LIN {X 0,Y 253.116,Z 526.81,A -85,B 0,C 180,E1 17086.147,E2 17086.147} C_VEL
LIN {X 0,Y 253.751,Z 526.81,A -85,B 0,C 180,E1 17093.136,E2 17093.136} C_VEL
LIN {X 0,Y 254.471,Z 526.81,A -85,B 0,C 180,E1 17099.989,E2 17099.989} C_VEL
LIN {X 0,Y 253.748,Z 526.81,A -85,B 0,C 180,E1 17106.843,E2 17106.843} C_VEL
LIN {X 0,Y 253.12,Z 526.81,A -85,B 0,C 180,E1 17113.832,E2 17113.832} C_VEL
LIN {X 0,Y 252.62,Z 526.81,A -85,B 0,C 180,E1 17121.064,E2 17121.064} C_VEL
LIN {X 0,Y 252.194,Z 526.81,A -85,B 0,C 180,E1 17128.69,E2 17128.69} C_VEL
LIN {X 0,Y 251.705,Z 526.81,A -85,B 0,C 180,E1 17136.964,E2 17136.964} C_VEL
LIN {X 0,Y 251.565,Z 526.81,A -85,B 0,C 180,E1 17146.221,E2 17146.221} C_VEL
LIN {X 0,Y 251.958,Z 526.81,A -85,B 0,C 180,E1 17150.844,E2 17150.844} C_VEL
LIN {X 0,Y 270.86,Z 591.901,A -85,B 0,C 180,E1 17154.954,E2 17154.954} C_VEL
LIN {X 0,Y 272.504,Z 601.249,A -85,B 0,C 180,E1 17155.665,E2 17155.665} C_VEL
LIN {X 0,Y 268.172,Z 634.394,A -85,B 0,C 180,E1 17158.572,E2 17158.572} C_VEL
LIN {X 0,Y 263.468,Z 664.052,A -85,B 0,C 180,E1 17162.639,E2 17162.639} C_VEL
LIN {X 0,Y 259.639,Z 689.343,A -85,B 0,C 180,E1 17167.736,E2 17167.736} C_VEL
LIN {X 0,Y 257.402,Z 710.001,A -85,B 0,C 180,E1 17173.784,E2 17173.784} C_VEL
LIN {X 0,Y 257.027,Z 723.846,A -85,B 0,C 180,E1 17179.829,E2 17179.829} C_VEL
LIN {X 0,Y 257.514,Z 731.331,A -85,B 0,C 180,E1 17184.948,E2 17184.948} C_VEL
LIN {X 0,Y 257.788,Z 735.161,A -85,B 0,C 180,E1 17190.008,E2 17190.008} C_VEL
LIN {X 0,Y 256.526,Z 734.875,A -85,B 0,C 180,E1 17196.787,E2 17196.787} C_VEL
LIN {X 0,Y 256.215,Z 728.457,A -85,B 0,C 180,E1 17204.554,E2 17204.554} C_VEL
LIN {X 0,Y 259.476,Z 716.032,A -85,B 0,C 180,E1 17212.298,E2 17212.298} C_VEL
LIN {X 0,Y 267.703,Z 697.17,A -85,B 0,C 180,E1 17219.671,E2 17219.671} C_VEL
LIN {X 0,Y 278.883,Z 674.315,A -85,B 0,C 180,E1 17225.604,E2 17225.604} C_VEL
LIN {X 0,Y 292.583,Z 646.621,A -85,B 0,C 180,E1 17230.314,E2 17230.314} C_VEL
LIN {X 0,Y 306.811,Z 613.528,A -85,B 0,C 180,E1 17234.03,E2 17234.03} C_VEL
LIN {X 0,Y 305.668,Z 605.43,A -85,B 0,C 180,E1 17237.281,E2 17237.281} C_VEL
LIN {X 0,Y 304.554,Z 603.17,A -85,B 0,C 180,E1 17239.752,E2 17239.752} C_VEL
LIN {X 0,Y 303.432,Z 604.168,A -85,B 0,C 180,E1 17243.231,E2 17243.231} C_VEL
LIN {X 0,Y 301.963,Z 610.894,A -85,B 0,C 180,E1 17246.944,E2 17246.944} C_VEL
LIN {X 0,Y 299.587,Z 618.107,A -85,B 0,C 180,E1 17248.987,E2 17248.987} C_VEL
LIN {X 0,Y 287.255,Z 640.013,A -85,B 0,C 180,E1 17253.395,E2 17253.395} C_VEL
LIN {X 0,Y 276.783,Z 655.626,A -85,B 0,C 180,E1 17258.428,E2 17258.428} C_VEL
LIN {X 0,Y 273.369,Z 659.975,A -85,B 0,C 180,E1 17260.458,E2 17260.458} C_VEL
LIN {X 0,Y 265.293,Z 666.359,A -85,B 0,C 180,E1 17263.486,E2 17263.486} C_VEL
LIN {X 0,Y 258.207,Z 669.931,A -85,B 0,C 180,E1 17266.346,E2 17266.346} C_VEL
LIN {X 0,Y 257.614,Z 670.127,A -85,B 0,C 180,E1 17266.81,E2 17266.81} C_VEL
LIN {X 0,Y 254.828,Z 671.039,A -85,B 0,C 180,E1 17269.744,E2 17269.744} C_VEL
LIN {X 0,Y 251.775,Z 669.41,A -85,B 0,C 180,E1 17274.836,E2 17274.836} C_VEL
LIN {X 0,Y 249.796,Z 662.54,A -85,B 0,C 180,E1 17280.912,E2 17280.912} C_VEL
LIN {X 0,Y 249.682,Z 649.701,A -85,B 0,C 180,E1 17286.976,E2 17286.976} C_VEL
LIN {X 0,Y 250.995,Z 630.908,A -85,B 0,C 180,E1 17292.641,E2 17292.641} C_VEL
LIN {X 0,Y 253.302,Z 607.549,A -85,B 0,C 180,E1 17297.4,E2 17297.4} C_VEL
LIN {X 0,Y 255.637,Z 580.367,A -85,B 0,C 180,E1 17301.17,E2 17301.17} C_VEL
LIN {X 0,Y 249.736,Z 549.406,A -85,B 0,C 180,E1 17304.37,E2 17304.37} C_VEL
LIN {X 0,Y 244.584,Z 526.81,A -85,B 0,C 180,E1 17306.183,E2 17306.183} C_VEL
LIN {X 0,Y 243.774,Z 526.81,A -85,B 0,C 180,E1 17316.141,E2 17316.141} C_VEL
LIN {X 0,Y 243.692,Z 526.81,A -85,B 0,C 180,E1 17323.125,E2 17323.125} C_VEL
LIN {X 0,Y 243.814,Z 526.81,A -85,B 0,C 180,E1 17331.601,E2 17331.601} C_VEL
LIN {X 0,Y 244.154,Z 526.81,A -85,B 0,C 180,E1 17340.265,E2 17340.265} C_VEL
LIN {X 0,Y 244.619,Z 526.81,A -85,B 0,C 180,E1 17348.212,E2 17348.212} C_VEL
LIN {X 0,Y 245.142,Z 526.81,A -85,B 0,C 180,E1 17355.688,E2 17355.688} C_VEL
LIN {X 0,Y 245.771,Z 526.81,A -85,B 0,C 180,E1 17362.914,E2 17362.914} C_VEL
LIN {X 0,Y 246.595,Z 526.81,A -85,B 0,C 180,E1 17369.992,E2 17369.992} C_VEL
LIN {X 0,Y 245.582,Z 526.81,A -85,B 0,C 180,E1 17379.399,E2 17379.399} C_VEL
LIN {X 0,Y 244.892,Z 526.81,A -85,B 0,C 180,E1 17387.998,E2 17387.998} C_VEL
LIN {X 0,Y 244.381,Z 526.81,A -85,B 0,C 180,E1 17395.692,E2 17395.692} C_VEL
LIN {X 0,Y 243.826,Z 526.81,A -85,B 0,C 180,E1 17403.967,E2 17403.967} C_VEL
LIN {X 0,Y 243.67,Z 526.81,A -85,B 0,C 180,E1 17413.106,E2 17413.106} C_VEL
LIN {X 0,Y 243.782,Z 526.81,A -85,B 0,C 180,E1 17421.594,E2 17421.594} C_VEL
LIN {X 0,Y 244.125,Z 526.81,A -85,B 0,C 180,E1 17430.243,E2 17430.243} C_VEL
LIN {X 0,Y 244.587,Z 526.81,A -85,B 0,C 180,E1 17438.186,E2 17438.186} C_VEL
LIN {X 0,Y 245.163,Z 526.81,A -85,B 0,C 180,E1 17445.688,E2 17445.688} C_VEL
LIN {X 0,Y 245.795,Z 526.81,A -85,B 0,C 180,E1 17452.913,E2 17452.913} C_VEL
LIN {X 0,Y 246.561,Z 526.81,A -85,B 0,C 180,E1 17459.989,E2 17459.989} C_VEL
LIN {X 0,Y 245.521,Z 526.81,A -85,B 0,C 180,E1 17469.413,E2 17469.413} C_VEL
LIN {X 0,Y 244.876,Z 526.81,A -85,B 0,C 180,E1 17477.996,E2 17477.996} C_VEL
LIN {X 0,Y 244.366,Z 526.81,A -85,B 0,C 180,E1 17485.69,E2 17485.69} C_VEL
LIN {X 0,Y 243.887,Z 526.81,A -85,B 0,C 180,E1 17493.953,E2 17493.953} C_VEL
LIN {X 0,Y 243.613,Z 526.81,A -85,B 0,C 180,E1 17503.112,E2 17503.112} C_VEL
LIN {X 0,Y 243.978,Z 526.81,A -85,B 0,C 180,E1 17510.328,E2 17510.328} C_VEL
LIN {X 0,Y 262.39,Z 590.644,A -85,B 0,C 180,E1 17514.439,E2 17514.439} C_VEL
LIN {X 0,Y 264.827,Z 601.026,A -85,B 0,C 180,E1 17515.279,E2 17515.279} C_VEL
LIN {X 0,Y 260.497,Z 633.255,A -85,B 0,C 180,E1 17518.198,E2 17518.198} C_VEL
LIN {X 0,Y 255.668,Z 663.218,A -85,B 0,C 180,E1 17522.425,E2 17522.425} C_VEL
LIN {X 0,Y 251.929,Z 687.654,A -85,B 0,C 180,E1 17527.481,E2 17527.481} C_VEL
LIN {X 0,Y 249.615,Z 708.493,A -85,B 0,C 180,E1 17533.716,E2 17533.716} C_VEL
LIN {X 0,Y 249.295,Z 723.223,A -85,B 0,C 180,E1 17540.394,E2 17540.394} C_VEL
LIN {X 0,Y 249.892,Z 731.257,A -85,B 0,C 180,E1 17546.535,E2 17546.535} C_VEL
LIN {X 0,Y 250.046,Z 733.566,A -85,B 0,C 180,E1 17550.008,E2 17550.008} C_VEL
LIN {X 0,Y 248.649,Z 733.566,A -85,B 0,C 180,E1 17557.003,E2 17557.003} C_VEL
LIN {X 0,Y 248.426,Z 727.533,A -85,B 0,C 180,E1 17565.021,E2 17565.021} C_VEL
LIN {X 0,Y 252.03,Z 715.545,A -85,B 0,C 180,E1 17572.994,E2 17572.994} C_VEL
LIN {X 0,Y 260.787,Z 697.428,A -85,B 0,C 180,E1 17580.54,E2 17580.54} C_VEL
LIN {X 0,Y 273.2,Z 674.491,A -85,B 0,C 180,E1 17586.794,E2 17586.794} C_VEL
LIN {X 0,Y 288.54,Z 646.199,A -85,B 0,C 180,E1 17591.75,E2 17591.75} C_VEL
LIN {X 0,Y 302.164,Z 617.648,A -85,B 0,C 180,E1 17595.064,E2 17595.064} C_VEL
LIN {X 0,Y 301.617,Z 612.201,A -85,B 0,C 180,E1 17597.46,E2 17597.46} C_VEL
LIN {X 0,Y 300.866,Z 610.491,A -85,B 0,C 180,E1 17599.155,E2 17599.155} C_VEL
LIN {X 0,Y 299.468,Z 610.666,A -85,B 0,C 180,E1 17602.662,E2 17602.662} C_VEL
LIN {X 0,Y 297.762,Z 615.675,A -85,B 0,C 180,E1 17606.003,E2 17606.003} C_VEL
LIN {X 0,Y 295.36,Z 621.611,A -85,B 0,C 180,E1 17607.883,E2 17607.883} C_VEL
LIN {X 0,Y 281.88,Z 643.133,A -85,B 0,C 180,E1 17612.414,E2 17612.414} C_VEL
LIN {X 0,Y 270.332,Z 658.41,A -85,B 0,C 180,E1 17617.671,E2 17617.671} C_VEL
LIN {X 0,Y 261.607,Z 667.374,A -85,B 0,C 180,E1 17623.191,E2 17623.191} C_VEL
LIN {X 0,Y 257.614,Z 670.127,A -85,B 0,C 180,E1 17626.81,E2 17626.81} C_VEL
LIN {X 0,Y 250.472,Z 671.806,A -85,B 0,C 180,E1 17630.393,E2 17630.393} C_VEL
LIN {X 0,Y 244.609,Z 671.157,A -85,B 0,C 180,E1 17633.65,E2 17633.65} C_VEL
LIN {X 0,Y 244.257,Z 670.821,A -85,B 0,C 180,E1 17634.149,E2 17634.149} C_VEL
LIN {X 0,Y 242.145,Z 664.48,A -85,B 0,C 180,E1 17640.011,E2 17640.011} C_VEL
LIN {X 0,Y 241.743,Z 651.942,A -85,B 0,C 180,E1 17646.303,E2 17646.303} C_VEL
LIN {X 0,Y 242.942,Z 633.679,A -85,B 0,C 180,E1 17652.153,E2 17652.153} C_VEL
LIN {X 0,Y 245.326,Z 609.376,A -85,B 0,C 180,E1 17657.362,E2 17657.362} C_VEL
LIN {X 0,Y 247.856,Z 581.525,A -85,B 0,C 180,E1 17661.394,E2 17661.394} C_VEL
LIN {X 0,Y 242.234,Z 551.6,A -85,B 0,C 180,E1 17664.615,E2 17664.615} C_VEL
LIN {X 0,Y 236.604,Z 526.81,A -85,B 0,C 180,E1 17666.623,E2 17666.623} C_VEL
LIN {X 0,Y 235.859,Z 526.81,A -85,B 0,C 180,E1 17675.304,E2 17675.304} C_VEL
LIN {X 0,Y 235.758,Z 526.81,A -85,B 0,C 180,E1 17679.969,E2 17679.969} C_VEL
LIN {X 0,Y 235.687,Z 526.81,A -85,B 0,C 180,E1 17685.025,E2 17685.025} C_VEL
LIN {X 0,Y 235.788,Z 526.81,A -85,B 0,C 180,E1 17690.418,E2 17690.418} C_VEL
LIN {X 0,Y 236.039,Z 526.81,A -85,B 0,C 180,E1 17699.115,E2 17699.115} C_VEL
LIN {X 0,Y 236.578,Z 526.81,A -85,B 0,C 180,E1 17707.409,E2 17707.409} C_VEL
LIN {X 0,Y 237.14,Z 526.81,A -85,B 0,C 180,E1 17715.194,E2 17715.194} C_VEL
LIN {X 0,Y 237.838,Z 526.81,A -85,B 0,C 180,E1 17722.677,E2 17722.677} C_VEL
LIN {X 0,Y 238.683,Z 526.81,A -85,B 0,C 180,E1 17729.991,E2 17729.991} C_VEL
LIN {X 0,Y 237.903,Z 526.81,A -85,B 0,C 180,E1 17737.304,E2 17737.304} C_VEL
LIN {X 0,Y 237,Z 526.81,A -85,B 0,C 180,E1 17746.581,E2 17746.581} C_VEL
LIN {X 0,Y 236.376,Z 526.81,A -85,B 0,C 180,E1 17756.247,E2 17756.247} C_VEL
LIN {X 0,Y 235.843,Z 526.81,A -85,B 0,C 180,E1 17765.284,E2 17765.284} C_VEL
LIN {X 0,Y 235.732,Z 526.81,A -85,B 0,C 180,E1 17769.951,E2 17769.951} C_VEL
LIN {X 0,Y 235.641,Z 526.81,A -85,B 0,C 180,E1 17775.013,E2 17775.013} C_VEL
LIN {X 0,Y 235.753,Z 526.81,A -85,B 0,C 180,E1 17780.4,E2 17780.4} C_VEL
LIN {X 0,Y 236.014,Z 526.81,A -85,B 0,C 180,E1 17789.111,E2 17789.111} C_VEL
LIN {X 0,Y 236.549,Z 526.81,A -85,B 0,C 180,E1 17797.405,E2 17797.405} C_VEL
LIN {X 0,Y 237.156,Z 526.81,A -85,B 0,C 180,E1 17805.194,E2 17805.194} C_VEL
LIN {X 0,Y 237.856,Z 526.81,A -85,B 0,C 180,E1 17812.675,E2 17812.675} C_VEL
LIN {X 0,Y 238.65,Z 526.81,A -85,B 0,C 180,E1 17819.989,E2 17819.989} C_VEL
LIN {X 0,Y 237.851,Z 526.81,A -85,B 0,C 180,E1 17827.303,E2 17827.303} C_VEL
LIN {X 0,Y 236.972,Z 526.81,A -85,B 0,C 180,E1 17836.619,E2 17836.619} C_VEL
LIN {X 0,Y 236.367,Z 526.81,A -85,B 0,C 180,E1 17846.282,E2 17846.282} C_VEL
LIN {X 0,Y 235.869,Z 526.81,A -85,B 0,C 180,E1 17855.274,E2 17855.274} C_VEL
LIN {X 0,Y 235.717,Z 526.81,A -85,B 0,C 180,E1 17859.948,E2 17859.948} C_VEL
LIN {X 0,Y 236.054,Z 527.414,A -85,B 0,C 180,E1 17869.796,E2 17869.796} C_VEL
LIN {X 0,Y 254.001,Z 589.667,A -85,B 0,C 180,E1 17873.938,E2 17873.938} C_VEL
LIN {X 0,Y 256.935,Z 602.437,A -85,B 0,C 180,E1 17875.009,E2 17875.009} C_VEL
LIN {X 0,Y 252.462,Z 634.482,A -85,B 0,C 180,E1 17878.105,E2 17878.105} C_VEL
LIN {X 0,Y 247.649,Z 663.805,A -85,B 0,C 180,E1 17882.485,E2 17882.485} C_VEL
LIN {X 0,Y 243.964,Z 687.652,A -85,B 0,C 180,E1 17887.668,E2 17887.668} C_VEL
LIN {X 0,Y 241.779,Z 708.126,A -85,B 0,C 180,E1 17894.108,E2 17894.108} C_VEL
LIN {X 0,Y 241.612,Z 722.544,A -85,B 0,C 180,E1 17900.995,E2 17900.995} C_VEL
LIN {X 0,Y 242.166,Z 729.412,A -85,B 0,C 180,E1 17906.424,E2 17906.424} C_VEL
LIN {X 0,Y 242.195,Z 732.019,A -85,B 0,C 180,E1 17910.32,E2 17910.32} C_VEL
LIN {X 0,Y 240.779,Z 732.236,A -85,B 0,C 180,E1 17917.233,E2 17917.233} C_VEL
LIN {X 0,Y 240.481,Z 727.454,A -85,B 0,C 180,E1 17924.595,E2 17924.595} C_VEL
LIN {X 0,Y 243.909,Z 716.681,A -85,B 0,C 180,E1 17932.837,E2 17932.837} C_VEL
LIN {X 0,Y 252.66,Z 700.014,A -85,B 0,C 180,E1 17940.631,E2 17940.631} C_VEL
LIN {X 0,Y 265.669,Z 678.147,A -85,B 0,C 180,E1 17947.257,E2 17947.257} C_VEL
LIN {X 0,Y 281.256,Z 652.198,A -85,B 0,C 180,E1 17952.301,E2 17952.301} C_VEL
LIN {X 0,Y 297.525,Z 622.132,A -85,B 0,C 180,E1 17956.037,E2 17956.037} C_VEL
LIN {X 0,Y 296.944,Z 617.891,A -85,B 0,C 180,E1 17958.497,E2 17958.497} C_VEL
LIN {X 0,Y 295.31,Z 617.241,A -85,B 0,C 180,E1 17962.044,E2 17962.044} C_VEL
LIN {X 0,Y 294.076,Z 619.565,A -85,B 0,C 180,E1 17964.432,E2 17964.432} C_VEL
LIN {X 0,Y 291.828,Z 624.383,A -85,B 0,C 180,E1 17966.558,E2 17966.558} C_VEL
LIN {X 0,Y 276.637,Z 646.313,A -85,B 0,C 180,E1 17971.399,E2 17971.399} C_VEL
LIN {X 0,Y 263.377,Z 661.863,A -85,B 0,C 180,E1 17977.18,E2 17977.18} C_VEL
LIN {X 0,Y 254.405,Z 669.729,A -85,B 0,C 180,E1 17982.7,E2 17982.7} C_VEL
LIN {X 0,Y 247.225,Z 672.621,A -85,B 0,C 180,E1 17989.425,E2 17989.425} C_VEL
LIN {X 0,Y 244.257,Z 670.821,A -85,B 0,C 180,E1 17994.149,E2 17994.149} C_VEL
LIN {X 0,Y 240.44,Z 668.494,A -85,B 0,C 180,E1 17997.074,E2 17997.074} C_VEL
LIN {X 0,Y 234.043,Z 662.72,A -85,B 0,C 180,E1 18001.393,E2 18001.393} C_VEL
LIN {X 0,Y 233.892,Z 661.818,A -85,B 0,C 180,E1 18001.886,E2 18001.886} C_VEL
LIN {X 0,Y 234.108,Z 646.79,A -85,B 0,C 180,E1 18008.378,E2 18008.378} C_VEL
LIN {X 0,Y 235.885,Z 625.302,A -85,B 0,C 180,E1 18014.413,E2 18014.413} C_VEL
LIN {X 0,Y 238.682,Z 598.201,A -85,B 0,C 180,E1 18019.464,E2 18019.464} C_VEL
LIN {X 0,Y 239.663,Z 580.078,A -85,B 0,C 180,E1 18021.919,E2 18021.919} C_VEL
LIN {X 0,Y 233.767,Z 549.81,A -85,B 0,C 180,E1 18025.2,E2 18025.2} C_VEL
LIN {X 0,Y 228.564,Z 526.81,A -85,B 0,C 180,E1 18027.075,E2 18027.075} C_VEL
LIN {X 0,Y 227.761,Z 526.81,A -85,B 0,C 180,E1 18037.073,E2 18037.073} C_VEL
LIN {X 0,Y 227.633,Z 526.81,A -85,B 0,C 180,E1 18047.039,E2 18047.039} C_VEL
LIN {X 0,Y 227.805,Z 526.81,A -85,B 0,C 180,E1 18053.25,E2 18053.25} C_VEL
LIN {X 0,Y 228.25,Z 526.81,A -85,B 0,C 180,E1 18062.323,E2 18062.323} C_VEL
LIN {X 0,Y 228.83,Z 526.81,A -85,B 0,C 180,E1 18070.671,E2 18070.671} C_VEL
LIN {X 0,Y 229.467,Z 526.81,A -85,B 0,C 180,E1 18078.574,E2 18078.574} C_VEL
LIN {X 0,Y 230.339,Z 526.81,A -85,B 0,C 180,E1 18086.222,E2 18086.222} C_VEL
LIN {X 0,Y 230.771,Z 526.81,A -85,B 0,C 180,E1 18089.991,E2 18089.991} C_VEL
LIN {X 0,Y 229.757,Z 526.81,A -85,B 0,C 180,E1 18098.647,E2 18098.647} C_VEL
LIN {X 0,Y 229.219,Z 526.81,A -85,B 0,C 180,E1 18105.311,E2 18105.311} C_VEL
LIN {X 0,Y 228.547,Z 526.81,A -85,B 0,C 180,E1 18113.411,E2 18113.411} C_VEL
LIN {X 0,Y 228.011,Z 526.81,A -85,B 0,C 180,E1 18122.078,E2 18122.078} C_VEL
LIN {X 0,Y 227.596,Z 526.81,A -85,B 0,C 180,E1 18131.689,E2 18131.689} C_VEL
LIN {X 0,Y 227.599,Z 526.81,A -85,B 0,C 180,E1 18138.287,E2 18138.287} C_VEL
LIN {X 0,Y 228.03,Z 526.81,A -85,B 0,C 180,E1 18147.903,E2 18147.903} C_VEL
LIN {X 0,Y 228.639,Z 526.81,A -85,B 0,C 180,E1 18157.962,E2 18157.962} C_VEL
LIN {X 0,Y 229.171,Z 526.81,A -85,B 0,C 180,E1 18164.665,E2 18164.665} C_VEL
LIN {X 0,Y 229.89,Z 526.81,A -85,B 0,C 180,E1 18172.42,E2 18172.42} C_VEL
LIN {X 0,Y 230.737,Z 526.81,A -85,B 0,C 180,E1 18179.988,E2 18179.988} C_VEL
LIN {X 0,Y 229.698,Z 526.81,A -85,B 0,C 180,E1 18188.668,E2 18188.668} C_VEL
LIN {X 0,Y 229.181,Z 526.81,A -85,B 0,C 180,E1 18195.31,E2 18195.31} C_VEL
LIN {X 0,Y 228.57,Z 526.81,A -85,B 0,C 180,E1 18203.405,E2 18203.405} C_VEL
LIN {X 0,Y 228.062,Z 526.81,A -85,B 0,C 180,E1 18212.065,E2 18212.065} C_VEL
LIN {X 0,Y 227.577,Z 526.81,A -85,B 0,C 180,E1 18221.687,E2 18221.687} C_VEL
LIN {X 0,Y 228.027,Z 527.128,A -85,B 0,C 180,E1 18229.188,E2 18229.188} C_VEL
LIN {X 0,Y 245.878,Z 589.566,A -85,B 0,C 180,E1 18233.502,E2 18233.502} C_VEL
LIN {X 0,Y 248.948,Z 604.366,A -85,B 0,C 180,E1 18234.8,E2 18234.8} C_VEL
LIN {X 0,Y 244.204,Z 637.001,A -85,B 0,C 180,E1 18238.207,E2 18238.207} C_VEL
LIN {X 0,Y 239.241,Z 666.623,A -85,B 0,C 180,E1 18243.004,E2 18243.004} C_VEL
LIN {X 0,Y 235.498,Z 691.165,A -85,B 0,C 180,E1 18248.889,E2 18248.889} C_VEL
LIN {X 0,Y 233.835,Z 709.815,A -85,B 0,C 180,E1 18255.424,E2 18255.424} C_VEL
LIN {X 0,Y 234.122,Z 723.122,A -85,B 0,C 180,E1 18262.577,E2 18262.577} C_VEL
LIN {X 0,Y 234.468,Z 729.027,A -85,B 0,C 180,E1 18268.159,E2 18268.159} C_VEL
LIN {X 0,Y 233.648,Z 731.198,A -85,B 0,C 180,E1 18273.724,E2 18273.724} C_VEL
LIN {X 0,Y 232.518,Z 729.191,A -85,B 0,C 180,E1 18281.274,E2 18281.274} C_VEL
LIN {X 0,Y 234.315,Z 721.136,A -85,B 0,C 180,E1 18290.077,E2 18290.077} C_VEL
LIN {X 0,Y 241.774,Z 706.72,A -85,B 0,C 180,E1 18298.779,E2 18298.779} C_VEL
LIN {X 0,Y 254.953,Z 686.263,A -85,B 0,C 180,E1 18306.442,E2 18306.442} C_VEL
LIN {X 0,Y 271.119,Z 662.206,A -85,B 0,C 180,E1 18312.088,E2 18312.088} C_VEL
LIN {X 0,Y 288.988,Z 633.302,A -85,B 0,C 180,E1 18316.368,E2 18316.368} C_VEL
LIN {X 0,Y 292.782,Z 626.559,A -85,B 0,C 180,E1 18317.136,E2 18317.136} C_VEL
LIN {X 0,Y 292.781,Z 625.361,A -85,B 0,C 180,E1 18317.772,E2 18317.772} C_VEL
LIN {X 0,Y 291.058,Z 623.729,A -85,B 0,C 180,E1 18321.388,E2 18321.388} C_VEL
LIN {X 0,Y 289.673,Z 625.406,A -85,B 0,C 180,E1 18323.833,E2 18323.833} C_VEL
LIN {X 0,Y 287.636,Z 628.846,A -85,B 0,C 180,E1 18325.549,E2 18325.549} C_VEL
LIN {X 0,Y 271.51,Z 649.614,A -85,B 0,C 180,E1 18330.349,E2 18330.349} C_VEL
LIN {X 0,Y 258.222,Z 663.596,A -85,B 0,C 180,E1 18335.78,E2 18335.78} C_VEL
LIN {X 0,Y 247.218,Z 672.025,A -85,B 0,C 180,E1 18342.181,E2 18342.181} C_VEL
LIN {X 0,Y 239.626,Z 674.161,A -85,B 0,C 180,E1 18349.085,E2 18349.085} C_VEL
LIN {X 0,Y 236.195,Z 671.458,A -85,B 0,C 180,E1 18354.494,E2 18354.494} C_VEL
LIN {X 0,Y 234.042,Z 663.473,A -85,B 0,C 180,E1 18360.938,E2 18360.938} C_VEL
LIN {X 0,Y 233.892,Z 661.818,A -85,B 0,C 180,E1 18361.886,E2 18361.886} C_VEL
LIN {X 0,Y 231.259,Z 656.211,A -85,B 0,C 180,E1 18364.735,E2 18364.735} C_VEL
LIN {X 0,Y 226.394,Z 645.901,A -85,B 0,C 180,E1 18368.82,E2 18368.82} C_VEL
LIN {X 0,Y 226.388,Z 644.569,A -85,B 0,C 180,E1 18369.266,E2 18369.266} C_VEL
LIN {X 0,Y 228.403,Z 621.878,A -85,B 0,C 180,E1 18375.388,E2 18375.388} C_VEL
LIN {X 0,Y 231.279,Z 594.459,A -85,B 0,C 180,E1 18380.342,E2 18380.342} C_VEL
LIN {X 0,Y 231.743,Z 580.114,A -85,B 0,C 180,E1 18382.278,E2 18382.278} C_VEL
LIN {X 0,Y 225.607,Z 548.844,A -85,B 0,C 180,E1 18385.746,E2 18385.746} C_VEL
LIN {X 0,Y 220.535,Z 526.81,A -85,B 0,C 180,E1 18387.623,E2 18387.623} C_VEL
LIN {X 0,Y 219.682,Z 526.81,A -85,B 0,C 180,E1 18398.35,E2 18398.35} C_VEL
LIN {X 0,Y 219.681,Z 526.81,A -85,B 0,C 180,E1 18406.419,E2 18406.419} C_VEL
LIN {X 0,Y 219.923,Z 526.81,A -85,B 0,C 180,E1 18416.569,E2 18416.569} C_VEL
LIN {X 0,Y 220.477,Z 526.81,A -85,B 0,C 180,E1 18425.657,E2 18425.657} C_VEL
LIN {X 0,Y 221.139,Z 526.81,A -85,B 0,C 180,E1 18434.096,E2 18434.096} C_VEL
LIN {X 0,Y 221.913,Z 526.81,A -85,B 0,C 180,E1 18442.148,E2 18442.148} C_VEL
LIN {X 0,Y 222.86,Z 526.81,A -85,B 0,C 180,E1 18449.991,E2 18449.991} C_VEL
LIN {X 0,Y 221.979,Z 526.81,A -85,B 0,C 180,E1 18457.831,E2 18457.831} C_VEL
LIN {X 0,Y 221.089,Z 526.81,A -85,B 0,C 180,E1 18466.481,E2 18466.481} C_VEL
LIN {X 0,Y 220.464,Z 526.81,A -85,B 0,C 180,E1 18474.324,E2 18474.324} C_VEL
LIN {X 0,Y 219.883,Z 526.81,A -85,B 0,C 180,E1 18483.415,E2 18483.415} C_VEL
LIN {X 0,Y 219.637,Z 526.81,A -85,B 0,C 180,E1 18493.566,E2 18493.566} C_VEL
LIN {X 0,Y 219.669,Z 526.81,A -85,B 0,C 180,E1 18501.647,E2 18501.647} C_VEL
LIN {X 0,Y 220.226,Z 526.81,A -85,B 0,C 180,E1 18511.22,E2 18511.22} C_VEL
LIN {X 0,Y 220.811,Z 526.81,A -85,B 0,C 180,E1 18519.938,E2 18519.938} C_VEL
LIN {X 0,Y 221.51,Z 526.81,A -85,B 0,C 180,E1 18528.155,E2 18528.155} C_VEL
LIN {X 0,Y 222.386,Z 526.81,A -85,B 0,C 180,E1 18536.084,E2 18536.084} C_VEL
LIN {X 0,Y 222.824,Z 526.81,A -85,B 0,C 180,E1 18539.988,E2 18539.988} C_VEL
LIN {X 0,Y 221.925,Z 526.81,A -85,B 0,C 180,E1 18547.83,E2 18547.83} C_VEL
LIN {X 0,Y 221.053,Z 526.81,A -85,B 0,C 180,E1 18556.515,E2 18556.515} C_VEL
LIN {X 0,Y 220.485,Z 526.81,A -85,B 0,C 180,E1 18564.317,E2 18564.317} C_VEL
LIN {X 0,Y 219.922,Z 526.81,A -85,B 0,C 180,E1 18573.403,E2 18573.403} C_VEL
LIN {X 0,Y 219.669,Z 526.81,A -85,B 0,C 180,E1 18583.551,E2 18583.551} C_VEL
LIN {X 0,Y 220.096,Z 527.488,A -85,B 0,C 180,E1 18588.605,E2 18588.605} C_VEL
LIN {X 0,Y 237.486,Z 588.809,A -85,B 0,C 180,E1 18593.004,E2 18593.004} C_VEL
LIN {X 0,Y 241.122,Z 604.698,A -85,B 0,C 180,E1 18594.474,E2 18594.474} C_VEL
LIN {X 0,Y 236.224,Z 637.621,A -85,B 0,C 180,E1 18598.087,E2 18598.087} C_VEL
LIN {X 0,Y 231.3,Z 666.5,A -85,B 0,C 180,E1 18603.002,E2 18603.002} C_VEL
LIN {X 0,Y 227.61,Z 690.841,A -85,B 0,C 180,E1 18609.122,E2 18609.122} C_VEL
LIN {X 0,Y 226.058,Z 708.95,A -85,B 0,C 180,E1 18615.768,E2 18615.768} C_VEL
LIN {X 0,Y 226.342,Z 720.896,A -85,B 0,C 180,E1 18622.321,E2 18622.321} C_VEL
LIN {X 0,Y 226.769,Z 727.201,A -85,B 0,C 180,E1 18628.096,E2 18628.096} C_VEL
LIN {X 0,Y 225.868,Z 729.555,A -85,B 0,C 180,E1 18633.853,E2 18633.853} C_VEL
LIN {X 0,Y 224.663,Z 727.936,A -85,B 0,C 180,E1 18641.674,E2 18641.674} C_VEL
LIN {X 0,Y 226.741,Z 720.256,A -85,B 0,C 180,E1 18650.836,E2 18650.836} C_VEL
LIN {X 0,Y 234.34,Z 707.289,A -85,B 0,C 180,E1 18659.393,E2 18659.393} C_VEL
LIN {X 0,Y 247.791,Z 688.458,A -85,B 0,C 180,E1 18667.123,E2 18667.123} C_VEL
LIN {X 0,Y 264.337,Z 666.188,A -85,B 0,C 180,E1 18672.868,E2 18672.868} C_VEL
LIN {X 0,Y 283.967,Z 637.636,A -85,B 0,C 180,E1 18677.441,E2 18677.441} C_VEL
LIN {X 0,Y 287.067,Z 632.84,A -85,B 0,C 180,E1 18677.991,E2 18677.991} C_VEL
LIN {X 0,Y 287.429,Z 631.197,A -85,B 0,C 180,E1 18678.775,E2 18678.775} C_VEL
LIN {X 0,Y 285.558,Z 630.713,A -85,B 0,C 180,E1 18682.697,E2 18682.697} C_VEL
LIN {X 0,Y 283.487,Z 633.411,A -85,B 0,C 180,E1 18684.505,E2 18684.505} C_VEL
LIN {X 0,Y 266.527,Z 653.009,A -85,B 0,C 180,E1 18689.265,E2 18689.265} C_VEL
LIN {X 0,Y 251.571,Z 666.819,A -85,B 0,C 180,E1 18695.097,E2 18695.097} C_VEL
LIN {X 0,Y 240.038,Z 674.3,A -85,B 0,C 180,E1 18701.629,E2 18701.629} C_VEL
LIN {X 0,Y 232.031,Z 675.59,A -85,B 0,C 180,E1 18708.723,E2 18708.723} C_VEL
LIN {X 0,Y 227.837,Z 671.197,A -85,B 0,C 180,E1 18715.535,E2 18715.535} C_VEL
LIN {X 0,Y 226.022,Z 662.078,A -85,B 0,C 180,E1 18721.931,E2 18721.931} C_VEL
LIN {X 0,Y 226.192,Z 647.732,A -85,B 0,C 180,E1 18728.189,E2 18728.189} C_VEL
LIN {X 0,Y 226.388,Z 644.569,A -85,B 0,C 180,E1 18729.266,E2 18729.266} C_VEL
LIN {X 0,Y 225.564,Z 639.136,A -85,B 0,C 180,E1 18730.989,E2 18730.989} C_VEL
LIN {X 0,Y 220.573,Z 622.715,A -85,B 0,C 180,E1 18735.399,E2 18735.399} C_VEL
LIN {X 0,Y 220.626,Z 621.03,A -85,B 0,C 180,E1 18735.771,E2 18735.771} C_VEL
LIN {X 0,Y 223.541,Z 594.095,A -85,B 0,C 180,E1 18740.698,E2 18740.698} C_VEL
LIN {X 0,Y 224.022,Z 581.606,A -85,B 0,C 180,E1 18742.447,E2 18742.447} C_VEL
LIN {X 0,Y 218.02,Z 550.801,A -85,B 0,C 180,E1 18746.007,E2 18746.007} C_VEL
LIN {X 0,Y 212.572,Z 526.81,A -85,B 0,C 180,E1 18748.105,E2 18748.105} C_VEL
LIN {X 0,Y 211.778,Z 526.81,A -85,B 0,C 180,E1 18758.132,E2 18758.132} C_VEL
LIN {X 0,Y 211.738,Z 526.81,A -85,B 0,C 180,E1 18765.664,E2 18765.664} C_VEL
LIN {X 0,Y 211.874,Z 526.81,A -85,B 0,C 180,E1 18775.12,E2 18775.12} C_VEL
LIN {X 0,Y 212.478,Z 526.81,A -85,B 0,C 180,E1 18784.677,E2 18784.677} C_VEL
LIN {X 0,Y 213.14,Z 526.81,A -85,B 0,C 180,E1 18793.482,E2 18793.482} C_VEL
LIN {X 0,Y 214.005,Z 526.81,A -85,B 0,C 180,E1 18802.162,E2 18802.162} C_VEL
LIN {X 0,Y 214.945,Z 526.81,A -85,B 0,C 180,E1 18809.99,E2 18809.99} C_VEL
LIN {X 0,Y 214,Z 526.81,A -85,B 0,C 180,E1 18818.125,E2 18818.125} C_VEL
LIN {X 0,Y 213.183,Z 526.81,A -85,B 0,C 180,E1 18826.494,E2 18826.494} C_VEL
LIN {X 0,Y 212.459,Z 526.81,A -85,B 0,C 180,E1 18835.304,E2 18835.304} C_VEL
LIN {X 0,Y 211.833,Z 526.81,A -85,B 0,C 180,E1 18844.864,E2 18844.864} C_VEL
LIN {X 0,Y 211.695,Z 526.81,A -85,B 0,C 180,E1 18854.324,E2 18854.324} C_VEL
LIN {X 0,Y 211.766,Z 526.81,A -85,B 0,C 180,E1 18861.841,E2 18861.841} C_VEL
LIN {X 0,Y 212.096,Z 526.81,A -85,B 0,C 180,E1 18870.007,E2 18870.007} C_VEL
LIN {X 0,Y 212.742,Z 526.81,A -85,B 0,C 180,E1 18879.142,E2 18879.142} C_VEL
LIN {X 0,Y 213.535,Z 526.81,A -85,B 0,C 180,E1 18887.706,E2 18887.706} C_VEL
LIN {X 0,Y 214.436,Z 526.81,A -85,B 0,C 180,E1 18895.939,E2 18895.939} C_VEL
LIN {X 0,Y 214.91,Z 526.81,A -85,B 0,C 180,E1 18899.988,E2 18899.988} C_VEL
LIN {X 0,Y 213.956,Z 526.81,A -85,B 0,C 180,E1 18908.123,E2 18908.123} C_VEL
LIN {X 0,Y 213.152,Z 526.81,A -85,B 0,C 180,E1 18916.493,E2 18916.493} C_VEL
LIN {X 0,Y 212.47,Z 526.81,A -85,B 0,C 180,E1 18925.298,E2 18925.298} C_VEL
LIN {X 0,Y 211.858,Z 526.81,A -85,B 0,C 180,E1 18934.854,E2 18934.854} C_VEL
LIN {X 0,Y 211.879,Z 526.81,A -85,B 0,C 180,E1 18945.589,E2 18945.589} C_VEL
LIN {X 0,Y 212.132,Z 526.81,A -85,B 0,C 180,E1 18947.924,E2 18947.924} C_VEL
LIN {X 0,Y 229.668,Z 589.719,A -85,B 0,C 180,E1 18952.652,E2 18952.652} C_VEL
LIN {X 0,Y 233.369,Z 604.49,A -85,B 0,C 180,E1 18954.107,E2 18954.107} C_VEL
LIN {X 0,Y 228.556,Z 636.319,A -85,B 0,C 180,E1 18957.728,E2 18957.728} C_VEL
LIN {X 0,Y 223.539,Z 665.29,A -85,B 0,C 180,E1 18962.804,E2 18962.804} C_VEL
LIN {X 0,Y 219.87,Z 689.002,A -85,B 0,C 180,E1 18968.935,E2 18968.935} C_VEL
LIN {X 0,Y 218.318,Z 707.896,A -85,B 0,C 180,E1 18976.085,E2 18976.085} C_VEL
LIN {X 0,Y 218.74,Z 719.964,A -85,B 0,C 180,E1 18983.052,E2 18983.052} C_VEL
LIN {X 0,Y 219.078,Z 725.231,A -85,B 0,C 180,E1 18988.029,E2 18988.029} C_VEL
LIN {X 0,Y 219.17,Z 726.58,A -85,B 0,C 180,E1 18990.009,E2 18990.009} C_VEL
LIN {X 0,Y 217.226,Z 727.878,A -85,B 0,C 180,E1 18998.023,E2 18998.023} C_VEL
LIN {X 0,Y 217.145,Z 724.235,A -85,B 0,C 180,E1 19006.205,E2 19006.205} C_VEL
LIN {X 0,Y 222.593,Z 713.797,A -85,B 0,C 180,E1 19016.25,E2 19016.25} C_VEL
LIN {X 0,Y 235.448,Z 696.936,A -85,B 0,C 180,E1 19025.374,E2 19025.374} C_VEL
LIN {X 0,Y 252.953,Z 675.607,A -85,B 0,C 180,E1 19032.339,E2 19032.339} C_VEL
LIN {X 0,Y 272.859,Z 650.343,A -85,B 0,C 180,E1 19037.338,E2 19037.338} C_VEL
LIN {X 0,Y 281.215,Z 638.829,A -85,B 0,C 180,E1 19038.928,E2 19038.928} C_VEL
LIN {X 0,Y 281.986,Z 636.85,A -85,B 0,C 180,E1 19039.9,E2 19039.9} C_VEL
LIN {X 0,Y 279.489,Z 638.04,A -85,B 0,C 180,E1 19043.437,E2 19043.437} C_VEL
LIN {X 0,Y 260.61,Z 657.395,A -85,B 0,C 180,E1 19048.489,E2 19048.489} C_VEL
LIN {X 0,Y 244.961,Z 669.992,A -85,B 0,C 180,E1 19054.377,E2 19054.377} C_VEL
LIN {X 0,Y 232.848,Z 676.482,A -85,B 0,C 180,E1 19061.04,E2 19061.04} C_VEL
LIN {X 0,Y 224.421,Z 677.006,A -85,B 0,C 180,E1 19068.336,E2 19068.336} C_VEL
LIN {X 0,Y 220.484,Z 673.022,A -85,B 0,C 180,E1 19074.298,E2 19074.298} C_VEL
LIN {X 0,Y 218.253,Z 663.987,A -85,B 0,C 180,E1 19081.006,E2 19081.006} C_VEL
LIN {X 0,Y 218.258,Z 648.54,A -85,B 0,C 180,E1 19087.987,E2 19087.987} C_VEL
LIN {X 0,Y 219.823,Z 628.727,A -85,B 0,C 180,E1 19093.961,E2 19093.961} C_VEL
LIN {X 0,Y 220.626,Z 621.03,A -85,B 0,C 180,E1 19095.771,E2 19095.771} C_VEL
LIN {X 0,Y 218.061,Z 607.633,A -85,B 0,C 180,E1 19098.601,E2 19098.601} C_VEL
LIN {X 0,Y 215.85,Z 593.004,A -85,B 0,C 180,E1 19101.168,E2 19101.168} C_VEL
LIN {X 0,Y 215.91,Z 580.617,A -85,B 0,C 180,E1 19102.937,E2 19102.937} C_VEL
LIN {X 0,Y 209.52,Z 548.569,A -85,B 0,C 180,E1 19106.692,E2 19106.692} C_VEL
LIN {X 0,Y 204.585,Z 526.81,A -85,B 0,C 180,E1 19108.673,E2 19108.673} C_VEL
LIN {X 0,Y 203.839,Z 526.81,A -85,B 0,C 180,E1 19116.471,E2 19116.471} C_VEL
LIN {X 0,Y 203.707,Z 526.81,A -85,B 0,C 180,E1 19122,E2 19122} C_VEL
LIN {X 0,Y 203.716,Z 526.81,A -85,B 0,C 180,E1 19128.023,E2 19128.023} C_VEL
LIN {X 0,Y 203.938,Z 526.81,A -85,B 0,C 180,E1 19134.77,E2 19134.77} C_VEL
LIN {X 0,Y 204.364,Z 526.81,A -85,B 0,C 180,E1 19143.596,E2 19143.596} C_VEL
LIN {X 0,Y 205.235,Z 526.81,A -85,B 0,C 180,E1 19153.581,E2 19153.581} C_VEL
LIN {X 0,Y 205.959,Z 526.81,A -85,B 0,C 180,E1 19161.535,E2 19161.535} C_VEL
LIN {X 0,Y 207.037,Z 526.81,A -85,B 0,C 180,E1 19169.99,E2 19169.99} C_VEL
LIN {X 0,Y 206.017,Z 526.81,A -85,B 0,C 180,E1 19178.442,E2 19178.442} C_VEL
LIN {X 0,Y 205.146,Z 526.81,A -85,B 0,C 180,E1 19187.16,E2 19187.16} C_VEL
LIN {X 0,Y 204.248,Z 526.81,A -85,B 0,C 180,E1 19197.161,E2 19197.161} C_VEL
LIN {X 0,Y 203.819,Z 526.81,A -85,B 0,C 180,E1 19206.449,E2 19206.449} C_VEL
LIN {X 0,Y 203.668,Z 526.81,A -85,B 0,C 180,E1 19211.981,E2 19211.981} C_VEL
LIN {X 0,Y 203.664,Z 526.81,A -85,B 0,C 180,E1 19218.008,E2 19218.008} C_VEL
LIN {X 0,Y 203.905,Z 526.81,A -85,B 0,C 180,E1 19224.747,E2 19224.747} C_VEL
LIN {X 0,Y 204.334,Z 526.81,A -85,B 0,C 180,E1 19233.59,E2 19233.59} C_VEL
LIN {X 0,Y 205.231,Z 526.81,A -85,B 0,C 180,E1 19243.513,E2 19243.513} C_VEL
LIN {X 0,Y 205.984,Z 526.81,A -85,B 0,C 180,E1 19252.155,E2 19252.155} C_VEL
LIN {X 0,Y 207,Z 526.81,A -85,B 0,C 180,E1 19259.987,E2 19259.987} C_VEL
LIN {X 0,Y 205.971,Z 526.81,A -85,B 0,C 180,E1 19268.441,E2 19268.441} C_VEL
LIN {X 0,Y 205.108,Z 526.81,A -85,B 0,C 180,E1 19277.159,E2 19277.159} C_VEL
LIN {X 0,Y 204.355,Z 526.81,A -85,B 0,C 180,E1 19286.378,E2 19286.378} C_VEL
LIN {X 0,Y 203.822,Z 526.81,A -85,B 0,C 180,E1 19296.442,E2 19296.442} C_VEL
LIN {X 0,Y 204.169,Z 526.85,A -85,B 0,C 180,E1 19307.341,E2 19307.341} C_VEL
LIN {X 0,Y 221.132,Z 588.427,A -85,B 0,C 180,E1 19312.102,E2 19312.102} C_VEL
LIN {X 0,Y 225.475,Z 605.331,A -85,B 0,C 180,E1 19313.835,E2 19313.835} C_VEL
LIN {X 0,Y 220.325,Z 638.156,A -85,B 0,C 180,E1 19317.831,E2 19317.831} C_VEL
LIN {X 0,Y 215.441,Z 666.22,A -85,B 0,C 180,E1 19323.112,E2 19323.112} C_VEL
LIN {X 0,Y 211.862,Z 689.75,A -85,B 0,C 180,E1 19329.621,E2 19329.621} C_VEL
LIN {X 0,Y 210.588,Z 707.049,A -85,B 0,C 180,E1 19336.561,E2 19336.561} C_VEL
LIN {X 0,Y 211.165,Z 718.965,A -85,B 0,C 180,E1 19343.836,E2 19343.836} C_VEL
LIN {X 0,Y 211.496,Z 724.682,A -85,B 0,C 180,E1 19350.01,E2 19350.01} C_VEL
LIN {X 0,Y 210.324,Z 726.175,A -85,B 0,C 180,E1 19354.138,E2 19354.138} C_VEL
LIN {X 0,Y 209.027,Z 725.239,A -85,B 0,C 180,E1 19362.561,E2 19362.561} C_VEL
LIN {X 0,Y 211.965,Z 718.144,A -85,B 0,C 180,E1 19372.921,E2 19372.921} C_VEL
LIN {X 0,Y 221.041,Z 706.45,A -85,B 0,C 180,E1 19381.827,E2 19381.827} C_VEL
LIN {X 0,Y 237.467,Z 688.113,A -85,B 0,C 180,E1 19390.219,E2 19390.219} C_VEL
LIN {X 0,Y 257.193,Z 666.318,A -85,B 0,C 180,E1 19396.16,E2 19396.16} C_VEL
LIN {X 0,Y 276.452,Z 643.15,A -85,B 0,C 180,E1 19400.074,E2 19400.074} C_VEL
LIN {X 0,Y 274.234,Z 644.049,A -85,B 0,C 180,E1 19402.619,E2 19402.619} C_VEL
LIN {X 0,Y 254.669,Z 661.721,A -85,B 0,C 180,E1 19407.666,E2 19407.666} C_VEL
LIN {X 0,Y 238.363,Z 673.11,A -85,B 0,C 180,E1 19413.614,E2 19413.614} C_VEL
LIN {X 0,Y 225.683,Z 678.622,A -85,B 0,C 180,E1 19420.414,E2 19420.414} C_VEL
LIN {X 0,Y 216.806,Z 678.271,A -85,B 0,C 180,E1 19427.92,E2 19427.92} C_VEL
LIN {X 0,Y 211.873,Z 671.716,A -85,B 0,C 180,E1 19435.915,E2 19435.915} C_VEL
LIN {X 0,Y 210.176,Z 659.109,A -85,B 0,C 180,E1 19443.627,E2 19443.627} C_VEL
LIN {X 0,Y 210.811,Z 641.869,A -85,B 0,C 180,E1 19450.356,E2 19450.356} C_VEL
LIN {X 0,Y 213.064,Z 618.623,A -85,B 0,C 180,E1 19456.526,E2 19456.526} C_VEL
LIN {X 0,Y 215.85,Z 593.004,A -85,B 0,C 180,E1 19461.168,E2 19461.168} C_VEL
LIN {X 0,Y 214.195,Z 583.731,A -85,B 0,C 180,E1 19462.603,E2 19462.603} C_VEL
LIN {X 0,Y 204.766,Z 563.55,A -85,B 0,C 180,E1 19465.549,E2 19465.549} C_VEL
LIN {X 0,Y 196.556,Z 526.81,A -85,B 0,C 180,E1 19469.195,E2 19469.195} C_VEL
LIN {X 0,Y 195.642,Z 526.81,A -85,B 0,C 180,E1 19479.278,E2 19479.278} C_VEL
LIN {X 0,Y 195.553,Z 526.81,A -85,B 0,C 180,E1 19485.813,E2 19485.813} C_VEL
LIN {X 0,Y 195.706,Z 526.81,A -85,B 0,C 180,E1 19491.75,E2 19491.75} C_VEL
LIN {X 0,Y 196.126,Z 526.81,A -85,B 0,C 180,E1 19498.144,E2 19498.144} C_VEL
LIN {X 0,Y 196.69,Z 526.81,A -85,B 0,C 180,E1 19507.506,E2 19507.506} C_VEL
LIN {X 0,Y 197.505,Z 526.81,A -85,B 0,C 180,E1 19516.693,E2 19516.693} C_VEL
LIN {X 0,Y 198.549,Z 526.81,A -85,B 0,C 180,E1 19525.616,E2 19525.616} C_VEL
LIN {X 0,Y 199.117,Z 526.81,A -85,B 0,C 180,E1 19529.99,E2 19529.99} C_VEL
LIN {X 0,Y 198.025,Z 526.81,A -85,B 0,C 180,E1 19538.785,E2 19538.785} C_VEL
LIN {X 0,Y 197.088,Z 526.81,A -85,B 0,C 180,E1 19547.885,E2 19547.885} C_VEL
LIN {X 0,Y 196.309,Z 526.81,A -85,B 0,C 180,E1 19557.554,E2 19557.554} C_VEL
LIN {X 0,Y 195.987,Z 526.81,A -85,B 0,C 180,E1 19562.724,E2 19562.724} C_VEL
LIN {X 0,Y 195.605,Z 526.81,A -85,B 0,C 180,E1 19569.264,E2 19569.264} C_VEL
LIN {X 0,Y 195.504,Z 526.81,A -85,B 0,C 180,E1 19575.797,E2 19575.797} C_VEL
LIN {X 0,Y 195.665,Z 526.81,A -85,B 0,C 180,E1 19581.739,E2 19581.739} C_VEL
LIN {X 0,Y 196.091,Z 526.81,A -85,B 0,C 180,E1 19588.12,E2 19588.12} C_VEL
LIN {X 0,Y 196.662,Z 526.81,A -85,B 0,C 180,E1 19597.47,E2 19597.47} C_VEL
LIN {X 0,Y 197.529,Z 526.81,A -85,B 0,C 180,E1 19606.693,E2 19606.693} C_VEL
LIN {X 0,Y 198.528,Z 526.81,A -85,B 0,C 180,E1 19615.613,E2 19615.613} C_VEL
LIN {X 0,Y 199.081,Z 526.81,A -85,B 0,C 180,E1 19619.987,E2 19619.987} C_VEL
LIN {X 0,Y 197.979,Z 526.81,A -85,B 0,C 180,E1 19628.784,E2 19628.784} C_VEL
LIN {X 0,Y 197.056,Z 526.81,A -85,B 0,C 180,E1 19637.884,E2 19637.884} C_VEL
LIN {X 0,Y 196.323,Z 526.81,A -85,B 0,C 180,E1 19647.546,E2 19647.546} C_VEL
LIN {X 0,Y 196.011,Z 526.81,A -85,B 0,C 180,E1 19652.714,E2 19652.714} C_VEL
LIN {X 0,Y 195.969,Z 526.81,A -85,B 0,C 180,E1 19664.033,E2 19664.033} C_VEL
LIN {X 0,Y 196.162,Z 526.81,A -85,B 0,C 180,E1 19666.63,E2 19666.63} C_VEL
LIN {X 0,Y 213.031,Z 588.527,A -85,B 0,C 180,E1 19671.683,E2 19671.683} C_VEL
LIN {X 0,Y 217.333,Z 607.645,A -85,B 0,C 180,E1 19673.726,E2 19673.726} C_VEL
LIN {X 0,Y 212.128,Z 639.654,A -85,B 0,C 180,E1 19677.948,E2 19677.948} C_VEL
LIN {X 0,Y 207.186,Z 668.07,A -85,B 0,C 180,E1 19683.713,E2 19683.713} C_VEL
LIN {X 0,Y 203.845,Z 690.68,A -85,B 0,C 180,E1 19690.484,E2 19690.484} C_VEL
LIN {X 0,Y 202.891,Z 708.131,A -85,B 0,C 180,E1 19698.168,E2 19698.168} C_VEL
LIN {X 0,Y 203.686,Z 719.119,A -85,B 0,C 180,E1 19705.747,E2 19705.747} C_VEL
LIN {X 0,Y 203.831,Z 722.702,A -85,B 0,C 180,E1 19710.01,E2 19710.01} C_VEL
LIN {X 0,Y 201.593,Z 724.664,A -85,B 0,C 180,E1 19718.649,E2 19718.649} C_VEL
LIN {X 0,Y 202.388,Z 720.586,A -85,B 0,C 180,E1 19729.573,E2 19729.573} C_VEL
LIN {X 0,Y 210.951,Z 709.828,A -85,B 0,C 180,E1 19740.569,E2 19740.569} C_VEL
LIN {X 0,Y 227.284,Z 693.352,A -85,B 0,C 180,E1 19749.794,E2 19749.794} C_VEL
LIN {X 0,Y 246.788,Z 674.077,A -85,B 0,C 180,E1 19756.139,E2 19756.139} C_VEL
LIN {X 0,Y 269.155,Z 650.278,A -85,B 0,C 180,E1 19760.823,E2 19760.823} C_VEL
LIN {X 0,Y 269.696,Z 649.365,A -85,B 0,C 180,E1 19761.366,E2 19761.366} C_VEL
LIN {X 0,Y 263.658,Z 654.492,A -85,B 0,C 180,E1 19762.932,E2 19762.932} C_VEL
LIN {X 0,Y 244.226,Z 669.005,A -85,B 0,C 180,E1 19768.215,E2 19768.215} C_VEL
LIN {X 0,Y 228.103,Z 677.759,A -85,B 0,C 180,E1 19774.455,E2 19774.455} C_VEL
LIN {X 0,Y 218.504,Z 680.653,A -85,B 0,C 180,E1 19779.743,E2 19779.743} C_VEL
LIN {X 0,Y 209.202,Z 679.505,A -85,B 0,C 180,E1 19787.474,E2 19787.474} C_VEL
LIN {X 0,Y 204.002,Z 672.125,A -85,B 0,C 180,E1 19795.757,E2 19795.757} C_VEL
LIN {X 0,Y 202.272,Z 658.859,A -85,B 0,C 180,E1 19803.768,E2 19803.768} C_VEL
LIN {X 0,Y 202.997,Z 640.838,A -85,B 0,C 180,E1 19810.759,E2 19810.759} C_VEL
LIN {X 0,Y 205.401,Z 616.516,A -85,B 0,C 180,E1 19817.161,E2 19817.161} C_VEL
LIN {X 0,Y 208.662,Z 587.82,A -85,B 0,C 180,E1 19822.266,E2 19822.266} C_VEL
LIN {X 0,Y 204.766,Z 563.55,A -85,B 0,C 180,E1 19825.549,E2 19825.549} C_VEL
LIN {X 0,Y 199.659,Z 552.432,A -85,B 0,C 180,E1 19826.947,E2 19826.947} C_VEL
LIN {X 0,Y 190.556,Z 536.022,A -85,B 0,C 180,E1 19828.851,E2 19828.851} C_VEL
LIN {X 0,Y 190.074,Z 533.965,A -85,B 0,C 180,E1 19829.033,E2 19829.033} C_VEL
LIN {X 0,Y 188.55,Z 526.81,A -85,B 0,C 180,E1 19829.696,E2 19829.696} C_VEL
LIN {X 0,Y 187.616,Z 526.81,A -85,B 0,C 180,E1 19840.227,E2 19840.227} C_VEL
LIN {X 0,Y 187.625,Z 526.81,A -85,B 0,C 180,E1 19849.777,E2 19849.777} C_VEL
LIN {X 0,Y 187.839,Z 526.81,A -85,B 0,C 180,E1 19855.638,E2 19855.638} C_VEL
LIN {X 0,Y 188.373,Z 526.81,A -85,B 0,C 180,E1 19862.17,E2 19862.17} C_VEL
LIN {X 0,Y 189.191,Z 526.81,A -85,B 0,C 180,E1 19873.85,E2 19873.85} C_VEL
LIN {X 0,Y 189.976,Z 526.81,A -85,B 0,C 180,E1 19880.817,E2 19880.817} C_VEL
LIN {X 0,Y 191.196,Z 526.81,A -85,B 0,C 180,E1 19889.989,E2 19889.989} C_VEL
LIN {X 0,Y 190.028,Z 526.81,A -85,B 0,C 180,E1 19899.158,E2 19899.158} C_VEL
LIN {X 0,Y 189.032,Z 526.81,A -85,B 0,C 180,E1 19908.675,E2 19908.675} C_VEL
LIN {X 0,Y 188.233,Z 526.81,A -85,B 0,C 180,E1 19918.844,E2 19918.844} C_VEL
LIN {X 0,Y 187.678,Z 526.81,A -85,B 0,C 180,E1 19926.202,E2 19926.202} C_VEL
LIN {X 0,Y 187.533,Z 526.81,A -85,B 0,C 180,E1 19936.588,E2 19936.588} C_VEL
LIN {X 0,Y 187.803,Z 526.81,A -85,B 0,C 180,E1 19945.628,E2 19945.628} C_VEL
LIN {X 0,Y 188.374,Z 526.81,A -85,B 0,C 180,E1 19952.121,E2 19952.121} C_VEL
LIN {X 0,Y 189.178,Z 526.81,A -85,B 0,C 180,E1 19963.785,E2 19963.785} C_VEL
LIN {X 0,Y 190.041,Z 526.81,A -85,B 0,C 180,E1 19972.26,E2 19972.26} C_VEL
LIN {X 0,Y 191.16,Z 526.81,A -85,B 0,C 180,E1 19979.986,E2 19979.986} C_VEL
LIN {X 0,Y 189.981,Z 526.81,A -85,B 0,C 180,E1 19989.157,E2 19989.157} C_VEL
LIN {X 0,Y 189.001,Z 526.81,A -85,B 0,C 180,E1 19998.673,E2 19998.673} C_VEL
LIN {X 0,Y 188.235,Z 526.81,A -85,B 0,C 180,E1 20008.838,E2 20008.838} C_VEL
LIN {X 0,Y 187.717,Z 526.81,A -85,B 0,C 180,E1 20020.164,E2 20020.164} C_VEL
LIN {X 0,Y 188.202,Z 526.81,A -85,B 0,C 180,E1 20025.976,E2 20025.976} C_VEL
LIN {X 0,Y 204.625,Z 587.647,A -85,B 0,C 180,E1 20031.166,E2 20031.166} C_VEL
LIN {X 0,Y 209.589,Z 607.203,A -85,B 0,C 180,E1 20033.356,E2 20033.356} C_VEL
LIN {X 0,Y 204.216,Z 639.437,A -85,B 0,C 180,E1 20037.811,E2 20037.811} C_VEL
LIN {X 0,Y 199.292,Z 667.546,A -85,B 0,C 180,E1 20043.796,E2 20043.796} C_VEL
LIN {X 0,Y 196.024,Z 689.969,A -85,B 0,C 180,E1 20050.848,E2 20050.848} C_VEL
LIN {X 0,Y 195.227,Z 707.197,A -85,B 0,C 180,E1 20058.831,E2 20058.831} C_VEL
LIN {X 0,Y 196.045,Z 716.738,A -85,B 0,C 180,E1 20065.581,E2 20065.581} C_VEL
LIN {X 0,Y 196.196,Z 720.596,A -85,B 0,C 180,E1 20070.01,E2 20070.01} C_VEL
LIN {X 0,Y 194.816,Z 722.448,A -85,B 0,C 180,E1 20074.468,E2 20074.468} C_VEL
LIN {X 0,Y 193.425,Z 722.258,A -85,B 0,C 180,E1 20083.593,E2 20083.593} C_VEL
LIN {X 0,Y 197.3,Z 716.222,A -85,B 0,C 180,E1 20094.977,E2 20094.977} C_VEL
LIN {X 0,Y 209.491,Z 704.505,A -85,B 0,C 180,E1 20105.335,E2 20105.335} C_VEL
LIN {X 0,Y 228.012,Z 688.154,A -85,B 0,C 180,E1 20113.558,E2 20113.558} C_VEL
LIN {X 0,Y 249.678,Z 668.593,A -85,B 0,C 180,E1 20119.302,E2 20119.302} C_VEL
LIN {X 0,Y 260.412,Z 658.048,A -85,B 0,C 180,E1 20121.567,E2 20121.567} C_VEL
LIN {X 0,Y 240.511,Z 671.429,A -85,B 0,C 180,E1 20126.591,E2 20126.591} C_VEL
LIN {X 0,Y 225.232,Z 679.042,A -85,B 0,C 180,E1 20131.944,E2 20131.944} C_VEL
LIN {X 0,Y 211.34,Z 682.607,A -85,B 0,C 180,E1 20139.025,E2 20139.025} C_VEL
LIN {X 0,Y 201.586,Z 680.569,A -85,B 0,C 180,E1 20146.992,E2 20146.992} C_VEL
LIN {X 0,Y 196.151,Z 672.479,A -85,B 0,C 180,E1 20155.587,E2 20155.587} C_VEL
LIN {X 0,Y 194.375,Z 658.4,A -85,B 0,C 180,E1 20163.922,E2 20163.922} C_VEL
LIN {X 0,Y 195.199,Z 639.658,A -85,B 0,C 180,E1 20171.195,E2 20171.195} C_VEL
LIN {X 0,Y 197.612,Z 615.656,A -85,B 0,C 180,E1 20177.553,E2 20177.553} C_VEL
LIN {X 0,Y 200.864,Z 586.258,A -85,B 0,C 180,E1 20182.829,E2 20182.829} C_VEL
LIN {X 0,Y 195.006,Z 555.414,A -85,B 0,C 180,E1 20186.924,E2 20186.924} C_VEL
LIN {X 0,Y 190.074,Z 533.965,A -85,B 0,C 180,E1 20189.033,E2 20189.033} C_VEL
LIN {X 0,Y 187.352,Z 528.356,A -85,B 0,C 180,E1 20190.546,E2 20190.546} C_VEL
LIN {X 0,Y 183.037,Z 526.194,A -85,B 0,C 180,E1 20193.64,E2 20193.64} C_VEL
LIN {X 0,Y 179.6,Z 526.81,A -85,B 0,C 180,E1 20199.005,E2 20199.005} C_VEL
LIN {X 0,Y 179.683,Z 526.81,A -85,B 0,C 180,E1 20209.34,E2 20209.34} C_VEL
LIN {X 0,Y 180.07,Z 526.81,A -85,B 0,C 180,E1 20219.689,E2 20219.689} C_VEL
LIN {X 0,Y 180.642,Z 526.81,A -85,B 0,C 180,E1 20227.248,E2 20227.248} C_VEL
LIN {X 0,Y 181.455,Z 526.81,A -85,B 0,C 180,E1 20235.492,E2 20235.492} C_VEL
LIN {X 0,Y 182.628,Z 526.81,A -85,B 0,C 180,E1 20245.233,E2 20245.233} C_VEL
LIN {X 0,Y 183.272,Z 526.81,A -85,B 0,C 180,E1 20249.989,E2 20249.989} C_VEL
LIN {X 0,Y 182.033,Z 526.81,A -85,B 0,C 180,E1 20259.564,E2 20259.564} C_VEL
LIN {X 0,Y 180.938,Z 526.81,A -85,B 0,C 180,E1 20269.543,E2 20269.543} C_VEL
LIN {X 0,Y 180.522,Z 526.81,A -85,B 0,C 180,E1 20274.782,E2 20274.782} C_VEL
LIN {X 0,Y 179.787,Z 526.81,A -85,B 0,C 180,E1 20286.107,E2 20286.107} C_VEL
LIN {X 0,Y 179.586,Z 526.81,A -85,B 0,C 180,E1 20297.57,E2 20297.57} C_VEL
LIN {X 0,Y 179.854,Z 526.81,A -85,B 0,C 180,E1 20307.313,E2 20307.313} C_VEL
LIN {X 0,Y 180.651,Z 526.81,A -85,B 0,C 180,E1 20317.181,E2 20317.181} C_VEL
LIN {X 0,Y 181.463,Z 526.81,A -85,B 0,C 180,E1 20325.49,E2 20325.49} C_VEL
LIN {X 0,Y 182.609,Z 526.81,A -85,B 0,C 180,E1 20335.23,E2 20335.23} C_VEL
LIN {X 0,Y 183.237,Z 526.81,A -85,B 0,C 180,E1 20339.985,E2 20339.985} C_VEL
LIN {X 0,Y 181.983,Z 526.81,A -85,B 0,C 180,E1 20349.563,E2 20349.563} C_VEL
LIN {X 0,Y 180.914,Z 526.81,A -85,B 0,C 180,E1 20359.541,E2 20359.541} C_VEL
LIN {X 0,Y 180.532,Z 526.81,A -85,B 0,C 180,E1 20364.775,E2 20364.775} C_VEL
LIN {X 0,Y 179.802,Z 526.81,A -85,B 0,C 180,E1 20376.098,E2 20376.098} C_VEL
LIN {X 0,Y 180.264,Z 526.81,A -85,B 0,C 180,E1 20385.331,E2 20385.331} C_VEL
LIN {X 0,Y 196.195,Z 586.827,A -85,B 0,C 180,E1 20390.647,E2 20390.647} C_VEL
LIN {X 0,Y 201.466,Z 608.723,A -85,B 0,C 180,E1 20393.224,E2 20393.224} C_VEL
LIN {X 0,Y 196.137,Z 640.028,A -85,B 0,C 180,E1 20397.843,E2 20397.843} C_VEL
LIN {X 0,Y 191.231,Z 668.054,A -85,B 0,C 180,E1 20404.197,E2 20404.197} C_VEL
LIN {X 0,Y 188.068,Z 690.637,A -85,B 0,C 180,E1 20411.835,E2 20411.835} C_VEL
LIN {X 0,Y 187.631,Z 706.187,A -85,B 0,C 180,E1 20419.55,E2 20419.55} C_VEL
LIN {X 0,Y 188.481,Z 715.493,A -85,B 0,C 180,E1 20426.557,E2 20426.557} C_VEL
LIN {X 0,Y 188.579,Z 718.453,A -85,B 0,C 180,E1 20430.011,E2 20430.011} C_VEL
LIN {X 0,Y 186.005,Z 721.12,A -85,B 0,C 180,E1 20439.381,E2 20439.381} C_VEL
LIN {X 0,Y 186.428,Z 719.173,A -85,B 0,C 180,E1 20448.969,E2 20448.969} C_VEL
LIN {X 0,Y 193.633,Z 711.995,A -85,B 0,C 180,E1 20459.976,E2 20459.976} C_VEL
LIN {X 0,Y 210.375,Z 698.612,A -85,B 0,C 180,E1 20470.383,E2 20470.383} C_VEL
LIN {X 0,Y 233.694,Z 680.195,A -85,B 0,C 180,E1 20478.178,E2 20478.178} C_VEL
LIN {X 0,Y 248.925,Z 667.484,A -85,B 0,C 180,E1 20481.454,E2 20481.454} C_VEL
LIN {X 0,Y 248.78,Z 667.278,A -85,B 0,C 180,E1 20481.975,E2 20481.975} C_VEL
LIN {X 0,Y 227.454,Z 678.544,A -85,B 0,C 180,E1 20487.839,E2 20487.839} C_VEL
LIN {X 0,Y 210.958,Z 683.797,A -85,B 0,C 180,E1 20494.508,E2 20494.508} C_VEL
LIN {X 0,Y 198.662,Z 683.71,A -85,B 0,C 180,E1 20502.266,E2 20502.266} C_VEL
LIN {X 0,Y 190.707,Z 677.911,A -85,B 0,C 180,E1 20510.878,E2 20510.878} C_VEL
LIN {X 0,Y 187.147,Z 667.568,A -85,B 0,C 180,E1 20518.855,E2 20518.855} C_VEL
LIN {X 0,Y 186.6,Z 651.153,A -85,B 0,C 180,E1 20527.005,E2 20527.005} C_VEL
LIN {X 0,Y 188.266,Z 629.389,A -85,B 0,C 180,E1 20534.3,E2 20534.3} C_VEL
LIN {X 0,Y 191.211,Z 603.379,A -85,B 0,C 180,E1 20540.283,E2 20540.283} C_VEL
LIN {X 0,Y 192.583,Z 584.045,A -85,B 0,C 180,E1 20543.515,E2 20543.515} C_VEL
LIN {X 0,Y 186.335,Z 552.302,A -85,B 0,C 180,E1 20547.76,E2 20547.76} C_VEL
LIN {X 0,Y 180.508,Z 526.81,A -85,B 0,C 180,E1 20550.454,E2 20550.454} C_VEL
LIN {X 0,Y 179.6,Z 526.81,A -85,B 0,C 180,E1 20559.005,E2 20559.005} C_VEL
LIN {X 0,Y 176.908,Z 526.81,A -85,B 0,C 180,E1 20563.123,E2 20563.123} C_VEL
LIN {X 0,Y 171.477,Z 526.81,A -85,B 0,C 180,E1 20570.216,E2 20570.216} C_VEL
LIN {X 0,Y 172.031,Z 526.81,A -85,B 0,C 180,E1 20578.111,E2 20578.111} C_VEL
LIN {X 0,Y 172.882,Z 526.81,A -85,B 0,C 180,E1 20589.481,E2 20589.481} C_VEL
LIN {X 0,Y 173.965,Z 526.81,A -85,B 0,C 180,E1 20599.964,E2 20599.964} C_VEL
LIN {X 0,Y 175.363,Z 526.81,A -85,B 0,C 180,E1 20609.988,E2 20609.988} C_VEL
LIN {X 0,Y 174.014,Z 526.81,A -85,B 0,C 180,E1 20620.009,E2 20620.009} C_VEL
LIN {X 0,Y 172.898,Z 526.81,A -85,B 0,C 180,E1 20630.492,E2 20630.492} C_VEL
LIN {X 0,Y 171.998,Z 526.81,A -85,B 0,C 180,E1 20641.868,E2 20641.868} C_VEL
LIN {X 0,Y 171.696,Z 526.81,A -85,B 0,C 180,E1 20648.103,E2 20648.103} C_VEL
LIN {X 0,Y 171.527,Z 526.81,A -85,B 0,C 180,E1 20655.058,E2 20655.058} C_VEL
LIN {X 0,Y 171.738,Z 526.81,A -85,B 0,C 180,E1 20662.49,E2 20662.49} C_VEL
LIN {X 0,Y 172.122,Z 526.81,A -85,B 0,C 180,E1 20671.575,E2 20671.575} C_VEL
LIN {X 0,Y 172.865,Z 526.81,A -85,B 0,C 180,E1 20679.476,E2 20679.476} C_VEL
LIN {X 0,Y 173.969,Z 526.81,A -85,B 0,C 180,E1 20689.961,E2 20689.961} C_VEL
LIN {X 0,Y 175.327,Z 526.81,A -85,B 0,C 180,E1 20699.985,E2 20699.985} C_VEL
LIN {X 0,Y 173.965,Z 526.81,A -85,B 0,C 180,E1 20710.008,E2 20710.008} C_VEL
LIN {X 0,Y 172.876,Z 526.81,A -85,B 0,C 180,E1 20720.49,E2 20720.49} C_VEL
LIN {X 0,Y 172.025,Z 526.81,A -85,B 0,C 180,E1 20731.856,E2 20731.856} C_VEL
LIN {X 0,Y 172.293,Z 526.81,A -85,B 0,C 180,E1 20744.645,E2 20744.645} C_VEL
LIN {X 0,Y 187.888,Z 586.246,A -85,B 0,C 180,E1 20750.151,E2 20750.151} C_VEL
LIN {X 0,Y 193.671,Z 608.33,A -85,B 0,C 180,E1 20752.886,E2 20752.886} C_VEL
LIN {X 0,Y 188.28,Z 639.424,A -85,B 0,C 180,E1 20757.694,E2 20757.694} C_VEL
LIN {X 0,Y 183.354,Z 667.287,A -85,B 0,C 180,E1 20764.321,E2 20764.321} C_VEL
LIN {X 0,Y 180.298,Z 689.69,A -85,B 0,C 180,E1 20772.289,E2 20772.289} C_VEL
LIN {X 0,Y 180.07,Z 705.093,A -85,B 0,C 180,E1 20780.33,E2 20780.33} C_VEL
LIN {X 0,Y 180.935,Z 714.161,A -85,B 0,C 180,E1 20787.613,E2 20787.613} C_VEL
LIN {X 0,Y 180.043,Z 717.376,A -85,B 0,C 180,E1 20792.421,E2 20792.421} C_VEL
LIN {X 0,Y 178.252,Z 719.215,A -85,B 0,C 180,E1 20799.793,E2 20799.793} C_VEL
LIN {X 0,Y 179.786,Z 716.792,A -85,B 0,C 180,E1 20812.172,E2 20812.172} C_VEL
LIN {X 0,Y 190.057,Z 708.86,A -85,B 0,C 180,E1 20823.906,E2 20823.906} C_VEL
LIN {X 0,Y 209.876,Z 695.087,A -85,B 0,C 180,E1 20834.038,E2 20834.038} C_VEL
LIN {X 0,Y 232.833,Z 678.769,A -85,B 0,C 180,E1 20840.566,E2 20840.566} C_VEL
LIN {X 0,Y 238.099,Z 674.851,A -85,B 0,C 180,E1 20841.664,E2 20841.664} C_VEL
LIN {X 0,Y 237.305,Z 674.931,A -85,B 0,C 180,E1 20842.359,E2 20842.359} C_VEL
LIN {X 0,Y 216.627,Z 683.29,A -85,B 0,C 180,E1 20848.402,E2 20848.402} C_VEL
LIN {X 0,Y 204.124,Z 685.976,A -85,B 0,C 180,E1 20853.59,E2 20853.59} C_VEL
LIN {X 0,Y 191.258,Z 684.97,A -85,B 0,C 180,E1 20861.555,E2 20861.555} C_VEL
LIN {X 0,Y 182.938,Z 678.347,A -85,B 0,C 180,E1 20870.487,E2 20870.487} C_VEL
LIN {X 0,Y 179.08,Z 666.312,A -85,B 0,C 180,E1 20879.409,E2 20879.409} C_VEL
LIN {X 0,Y 178.8,Z 648.567,A -85,B 0,C 180,E1 20887.924,E2 20887.924} C_VEL
LIN {X 0,Y 180.713,Z 626.19,A -85,B 0,C 180,E1 20895.251,E2 20895.251} C_VEL
LIN {X 0,Y 183.949,Z 598.562,A -85,B 0,C 180,E1 20901.437,E2 20901.437} C_VEL
LIN {X 0,Y 184.528,Z 583.881,A -85,B 0,C 180,E1 20903.914,E2 20903.914} C_VEL
LIN {X 0,Y 178.494,Z 552.978,A -85,B 0,C 180,E1 20908.181,E2 20908.181} C_VEL
LIN {X 0,Y 172.513,Z 526.81,A -85,B 0,C 180,E1 20911.041,E2 20911.041} C_VEL
LIN {X 0,Y 171.601,Z 526.81,A -85,B 0,C 180,E1 20918.867,E2 20918.867} C_VEL
LIN {X 0,Y 171.578,Z 526.81,A -85,B 0,C 180,E1 20925.077,E2 20925.077} C_VEL
LIN {X 0,Y 171.477,Z 526.81,A -85,B 0,C 180,E1 20930.216,E2 20930.216} C_VEL
LIN {X 0,Y 169.146,Z 526.81,A -85,B 0,C 180,E1 20934.542,E2 20934.542} C_VEL
LIN {X 0,Y 164.19,Z 526.81,A -85,B 0,C 180,E1 20942.002,E2 20942.002} C_VEL
LIN {X 0,Y 164.743,Z 526.81,A -85,B 0,C 180,E1 20948.418,E2 20948.418} C_VEL
LIN {X 0,Y 165.946,Z 526.81,A -85,B 0,C 180,E1 20959.473,E2 20959.473} C_VEL
LIN {X 0,Y 167.433,Z 526.81,A -85,B 0,C 180,E1 20969.988,E2 20969.988} C_VEL
LIN {X 0,Y 165.992,Z 526.81,A -85,B 0,C 180,E1 20980.499,E2 20980.499} C_VEL
LIN {X 0,Y 164.754,Z 526.81,A -85,B 0,C 180,E1 20991.554,E2 20991.554} C_VEL
LIN {X 0,Y 164.291,Z 526.81,A -85,B 0,C 180,E1 20997.424,E2 20997.424} C_VEL
LIN {X 0,Y 163.832,Z 526.81,A -85,B 0,C 180,E1 21003.697,E2 21003.697} C_VEL
LIN {X 0,Y 163.426,Z 526.81,A -85,B 0,C 180,E1 21012.148,E2 21012.148} C_VEL
LIN {X 0,Y 163.465,Z 526.81,A -85,B 0,C 180,E1 21019.563,E2 21019.563} C_VEL
LIN {X 0,Y 163.839,Z 526.81,A -85,B 0,C 180,E1 21026.308,E2 21026.308} C_VEL
LIN {X 0,Y 164.52,Z 526.81,A -85,B 0,C 180,E1 21036.937,E2 21036.937} C_VEL
LIN {X 0,Y 165.333,Z 526.81,A -85,B 0,C 180,E1 21044.038,E2 21044.038} C_VEL
LIN {X 0,Y 166.689,Z 526.81,A -85,B 0,C 180,E1 21054.773,E2 21054.773} C_VEL
LIN {X 0,Y 167.398,Z 526.81,A -85,B 0,C 180,E1 21059.984,E2 21059.984} C_VEL
LIN {X 0,Y 165.942,Z 526.81,A -85,B 0,C 180,E1 21070.497,E2 21070.497} C_VEL
LIN {X 0,Y 164.739,Z 526.81,A -85,B 0,C 180,E1 21081.551,E2 21081.551} C_VEL
LIN {X 0,Y 164.293,Z 526.81,A -85,B 0,C 180,E1 21087.418,E2 21087.418} C_VEL
LIN {X 0,Y 163.88,Z 526.81,A -85,B 0,C 180,E1 21093.77,E2 21093.77} C_VEL
LIN {X 0,Y 164.216,Z 526.81,A -85,B 0,C 180,E1 21103.914,E2 21103.914} C_VEL
LIN {X 0,Y 179.837,Z 586.472,A -85,B 0,C 180,E1 21109.744,E2 21109.744} C_VEL
LIN {X 0,Y 185.699,Z 608.831,A -85,B 0,C 180,E1 21112.667,E2 21112.667} C_VEL
LIN {X 0,Y 180.241,Z 639.748,A -85,B 0,C 180,E1 21117.758,E2 21117.758} C_VEL
LIN {X 0,Y 175.49,Z 666.386,A -85,B 0,C 180,E1 21124.458,E2 21124.458} C_VEL
LIN {X 0,Y 172.579,Z 688.659,A -85,B 0,C 180,E1 21132.789,E2 21132.789} C_VEL
LIN {X 0,Y 172.537,Z 703.906,A -85,B 0,C 180,E1 21141.178,E2 21141.178} C_VEL
LIN {X 0,Y 173.383,Z 712.729,A -85,B 0,C 180,E1 21148.761,E2 21148.761} C_VEL
LIN {X 0,Y 171.709,Z 716.133,A -85,B 0,C 180,E1 21155.071,E2 21155.071} C_VEL
LIN {X 0,Y 170.282,Z 717.154,A -85,B 0,C 180,E1 21165.483,E2 21165.483} C_VEL
LIN {X 0,Y 175.66,Z 713.044,A -85,B 0,C 180,E1 21178.312,E2 21178.312} C_VEL
LIN {X 0,Y 192.293,Z 702.86,A -85,B 0,C 180,E1 21190.524,E2 21190.524} C_VEL
LIN {X 0,Y 215.461,Z 688.586,A -85,B 0,C 180,E1 21199.076,E2 21199.076} C_VEL
LIN {X 0,Y 227.265,Z 680.997,A -85,B 0,C 180,E1 21201.909,E2 21201.909} C_VEL
LIN {X 0,Y 225.426,Z 681.449,A -85,B 0,C 180,E1 21202.826,E2 21202.826} C_VEL
LIN {X 0,Y 205.752,Z 687.084,A -85,B 0,C 180,E1 21209.012,E2 21209.012} C_VEL
LIN {X 0,Y 189.953,Z 687.785,A -85,B 0,C 180,E1 21216.53,E2 21216.53} C_VEL
LIN {X 0,Y 178.769,Z 683.165,A -85,B 0,C 180,E1 21225.297,E2 21225.297} C_VEL
LIN {X 0,Y 172.534,Z 672.581,A -85,B 0,C 180,E1 21234.981,E2 21234.981} C_VEL
LIN {X 0,Y 170.72,Z 656.148,A -85,B 0,C 180,E1 21244.466,E2 21244.466} C_VEL
LIN {X 0,Y 172.002,Z 633.799,A -85,B 0,C 180,E1 21253.052,E2 21253.052} C_VEL
LIN {X 0,Y 174.97,Z 607.351,A -85,B 0,C 180,E1 21259.936,E2 21259.936} C_VEL
LIN {X 0,Y 176.919,Z 586.006,A -85,B 0,C 180,E1 21263.91,E2 21263.91} C_VEL
LIN {X 0,Y 170.854,Z 554.776,A -85,B 0,C 180,E1 21268.471,E2 21268.471} C_VEL
LIN {X 0,Y 164.5,Z 526.81,A -85,B 0,C 180,E1 21271.593,E2 21271.593} C_VEL
LIN {X 0,Y 163.473,Z 526.81,A -85,B 0,C 180,E1 21282.169,E2 21282.169} C_VEL
LIN {X 0,Y 163.458,Z 526.81,A -85,B 0,C 180,E1 21290.135,E2 21290.135} C_VEL
LIN {X 0,Y 163.875,Z 526.81,A -85,B 0,C 180,E1 21296.319,E2 21296.319} C_VEL
LIN {X 0,Y 164.19,Z 526.81,A -85,B 0,C 180,E1 21302.002,E2 21302.002} C_VEL
LIN {X 0,Y 162.416,Z 526.81,A -85,B 0,C 180,E1 21306.523,E2 21306.523} C_VEL
LIN {X 0,Y 157.451,Z 526.81,A -85,B 0,C 180,E1 21314.315,E2 21314.315} C_VEL
LIN {X 0,Y 158.693,Z 526.81,A -85,B 0,C 180,E1 21324.512,E2 21324.512} C_VEL
LIN {X 0,Y 159.505,Z 526.81,A -85,B 0,C 180,E1 21329.987,E2 21329.987} C_VEL
LIN {X 0,Y 157.942,Z 526.81,A -85,B 0,C 180,E1 21341.04,E2 21341.04} C_VEL
LIN {X 0,Y 157.282,Z 526.81,A -85,B 0,C 180,E1 21346.772,E2 21346.772} C_VEL
LIN {X 0,Y 156.688,Z 526.81,A -85,B 0,C 180,E1 21352.724,E2 21352.724} C_VEL
LIN {X 0,Y 156.086,Z 526.81,A -85,B 0,C 180,E1 21359.159,E2 21359.159} C_VEL
LIN {X 0,Y 155.476,Z 526.81,A -85,B 0,C 180,E1 21368.801,E2 21368.801} C_VEL
LIN {X 0,Y 155.476,Z 526.81,A -85,B 0,C 180,E1 21381.154,E2 21381.154} C_VEL
LIN {X 0,Y 156.106,Z 526.81,A -85,B 0,C 180,E1 21390.973,E2 21390.973} C_VEL
LIN {X 0,Y 156.662,Z 526.81,A -85,B 0,C 180,E1 21397.241,E2 21397.241} C_VEL
LIN {X 0,Y 157.434,Z 526.81,A -85,B 0,C 180,E1 21404.047,E2 21404.047} C_VEL
LIN {X 0,Y 158.687,Z 526.81,A -85,B 0,C 180,E1 21414.508,E2 21414.508} C_VEL
LIN {X 0,Y 159.489,Z 526.81,A -85,B 0,C 180,E1 21419.983,E2 21419.983} C_VEL
LIN {X 0,Y 157.894,Z 526.81,A -85,B 0,C 180,E1 21431.039,E2 21431.039} C_VEL
LIN {X 0,Y 157.239,Z 526.81,A -85,B 0,C 180,E1 21436.772,E2 21436.772} C_VEL
LIN {X 0,Y 156.7,Z 526.81,A -85,B 0,C 180,E1 21442.716,E2 21442.716} C_VEL
LIN {X 0,Y 156.093,Z 526.81,A -85,B 0,C 180,E1 21449.22,E2 21449.22} C_VEL
LIN {X 0,Y 156.173,Z 526.81,A -85,B 0,C 180,E1 21463.145,E2 21463.145} C_VEL
LIN {X 0,Y 171.617,Z 586.131,A -85,B 0,C 180,E1 21469.276,E2 21469.276} C_VEL
LIN {X 0,Y 177.705,Z 609.556,A -85,B 0,C 180,E1 21472.499,E2 21472.499} C_VEL
LIN {X 0,Y 172.221,Z 639.784,A -85,B 0,C 180,E1 21477.815,E2 21477.815} C_VEL
LIN {X 0,Y 167.403,Z 666.987,A -85,B 0,C 180,E1 21485.162,E2 21485.162} C_VEL
LIN {X 0,Y 164.821,Z 688.895,A -85,B 0,C 180,E1 21494.016,E2 21494.016} C_VEL
LIN {X 0,Y 165.239,Z 704.425,A -85,B 0,C 180,E1 21503.436,E2 21503.436} C_VEL
LIN {X 0,Y 165.917,Z 711.222,A -85,B 0,C 180,E1 21510.012,E2 21510.012} C_VEL
LIN {X 0,Y 162.826,Z 715.067,A -85,B 0,C 180,E1 21520.731,E2 21520.731} C_VEL
LIN {X 0,Y 164.358,Z 714.195,A -85,B 0,C 180,E1 21532.947,E2 21532.947} C_VEL
LIN {X 0,Y 176.948,Z 707.421,A -85,B 0,C 180,E1 21546.81,E2 21546.81} C_VEL
LIN {X 0,Y 199.72,Z 695.397,A -85,B 0,C 180,E1 21557.513,E2 21557.513} C_VEL
LIN {X 0,Y 215.009,Z 686.892,A -85,B 0,C 180,E1 21561.841,E2 21561.841} C_VEL
LIN {X 0,Y 216.245,Z 685.927,A -85,B 0,C 180,E1 21562.573,E2 21562.573} C_VEL
LIN {X 0,Y 199.317,Z 689.466,A -85,B 0,C 180,E1 21567.895,E2 21567.895} C_VEL
LIN {X 0,Y 182.869,Z 689.2,A -85,B 0,C 180,E1 21575.563,E2 21575.563} C_VEL
LIN {X 0,Y 171.164,Z 683.713,A -85,B 0,C 180,E1 21584.628,E2 21584.628} C_VEL
LIN {X 0,Y 164.682,Z 672.359,A -85,B 0,C 180,E1 21594.741,E2 21594.741} C_VEL
LIN {X 0,Y 162.85,Z 655.011,A -85,B 0,C 180,E1 21604.682,E2 21604.682} C_VEL
LIN {X 0,Y 164.122,Z 633.308,A -85,B 0,C 180,E1 21613.139,E2 21613.139} C_VEL
LIN {X 0,Y 167.13,Z 606.909,A -85,B 0,C 180,E1 21620.221,E2 21620.221} C_VEL
LIN {X 0,Y 169.099,Z 587.055,A -85,B 0,C 180,E1 21624.059,E2 21624.059} C_VEL
LIN {X 0,Y 163.021,Z 555.509,A -85,B 0,C 180,E1 21628.889,E2 21628.889} C_VEL
LIN {X 0,Y 156.412,Z 526.81,A -85,B 0,C 180,E1 21632.389,E2 21632.389} C_VEL
LIN {X 0,Y 155.494,Z 526.81,A -85,B 0,C 180,E1 21642.99,E2 21642.99} C_VEL
LIN {X 0,Y 155.651,Z 526.81,A -85,B 0,C 180,E1 21654.277,E2 21654.277} C_VEL
LIN {X 0,Y 156.08,Z 526.81,A -85,B 0,C 180,E1 21661.991,E2 21661.991} C_VEL
LIN {X 0,Y 156.685,Z 526.81,A -85,B 0,C 180,E1 21667.247,E2 21667.247} C_VEL
LIN {X 0,Y 157.451,Z 526.81,A -85,B 0,C 180,E1 21674.315,E2 21674.315} C_VEL
LIN {X 0,Y 155.185,Z 526.81,A -85,B 0,C 180,E1 21679.038,E2 21679.038} C_VEL
LIN {X 0,Y 150.954,Z 526.81,A -85,B 0,C 180,E1 21687.181,E2 21687.181} C_VEL
LIN {X 0,Y 151.451,Z 526.81,A -85,B 0,C 180,E1 21690.485,E2 21690.485} C_VEL
LIN {X 0,Y 149.917,Z 526.81,A -85,B 0,C 180,E1 21701.639,E2 21701.639} C_VEL
LIN {X 0,Y 148.614,Z 526.81,A -85,B 0,C 180,E1 21713.483,E2 21713.483} C_VEL
LIN {X 0,Y 147.656,Z 526.81,A -85,B 0,C 180,E1 21724.856,E2 21724.856} C_VEL
LIN {X 0,Y 147.48,Z 526.81,A -85,B 0,C 180,E1 21735.922,E2 21735.922} C_VEL
LIN {X 0,Y 147.655,Z 526.81,A -85,B 0,C 180,E1 21745.093,E2 21745.093} C_VEL
LIN {X 0,Y 148.6,Z 526.81,A -85,B 0,C 180,E1 21756.456,E2 21756.456} C_VEL
LIN {X 0,Y 149.871,Z 526.81,A -85,B 0,C 180,E1 21768.326,E2 21768.326} C_VEL
LIN {X 0,Y 151.57,Z 526.81,A -85,B 0,C 180,E1 21779.982,E2 21779.982} C_VEL
LIN {X 0,Y 149.871,Z 526.81,A -85,B 0,C 180,E1 21791.638,E2 21791.638} C_VEL
LIN {X 0,Y 148.499,Z 526.81,A -85,B 0,C 180,E1 21804.048,E2 21804.048} C_VEL
LIN {X 0,Y 147.819,Z 526.81,A -85,B 0,C 180,E1 21814.998,E2 21814.998} C_VEL
LIN {X 0,Y 148.154,Z 526.81,A -85,B 0,C 180,E1 21822.422,E2 21822.422} C_VEL
LIN {X 0,Y 163.378,Z 585.86,A -85,B 0,C 180,E1 21828.819,E2 21828.819} C_VEL
LIN {X 0,Y 169.689,Z 610.322,A -85,B 0,C 180,E1 21832.369,E2 21832.369} C_VEL
LIN {X 0,Y 163.921,Z 641.445,A -85,B 0,C 180,E1 21838.324,E2 21838.324} C_VEL
LIN {X 0,Y 159.219,Z 668.223,A -85,B 0,C 180,E1 21846.221,E2 21846.221} C_VEL
LIN {X 0,Y 157.122,Z 688.771,A -85,B 0,C 180,E1 21855.243,E2 21855.243} C_VEL
LIN {X 0,Y 157.857,Z 703.048,A -85,B 0,C 180,E1 21864.509,E2 21864.509} C_VEL
LIN {X 0,Y 158.417,Z 708.598,A -85,B 0,C 180,E1 21870.013,E2 21870.013} C_VEL
LIN {X 0,Y 155.179,Z 712.815,A -85,B 0,C 180,E1 21881.266,E2 21881.266} C_VEL
LIN {X 0,Y 156.479,Z 712.687,A -85,B 0,C 180,E1 21892.784,E2 21892.784} C_VEL
LIN {X 0,Y 167.234,Z 707.986,A -85,B 0,C 180,E1 21906.064,E2 21906.064} C_VEL
LIN {X 0,Y 189.678,Z 697.916,A -85,B 0,C 180,E1 21917.608,E2 21917.608} C_VEL
LIN {X 0,Y 204.674,Z 690.694,A -85,B 0,C 180,E1 21922.164,E2 21922.164} C_VEL
LIN {X 0,Y 205.401,Z 690.135,A -85,B 0,C 180,E1 21922.702,E2 21922.702} C_VEL
LIN {X 0,Y 183.822,Z 691.716,A -85,B 0,C 180,E1 21930.402,E2 21930.402} C_VEL
LIN {X 0,Y 169.185,Z 687.988,A -85,B 0,C 180,E1 21939.043,E2 21939.043} C_VEL
LIN {X 0,Y 159.619,Z 678.808,A -85,B 0,C 180,E1 21949.082,E2 21949.082} C_VEL
LIN {X 0,Y 155.403,Z 664.337,A -85,B 0,C 180,E1 21959.319,E2 21959.319} C_VEL
LIN {X 0,Y 155.24,Z 645.742,A -85,B 0,C 180,E1 21968.429,E2 21968.429} C_VEL
LIN {X 0,Y 157.643,Z 619.91,A -85,B 0,C 180,E1 21977.123,E2 21977.123} C_VEL
LIN {X 0,Y 161.452,Z 589.358,A -85,B 0,C 180,E1 21983.956,E2 21983.956} C_VEL
LIN {X 0,Y 155.392,Z 557.295,A -85,B 0,C 180,E1 21989.173,E2 21989.173} C_VEL
LIN {X 0,Y 148.382,Z 526.81,A -85,B 0,C 180,E1 21992.947,E2 21992.947} C_VEL
LIN {X 0,Y 147.529,Z 526.81,A -85,B 0,C 180,E1 22005.946,E2 22005.946} C_VEL
LIN {X 0,Y 147.694,Z 526.81,A -85,B 0,C 180,E1 22015.123,E2 22015.123} C_VEL
LIN {X 0,Y 148.602,Z 526.81,A -85,B 0,C 180,E1 22026.528,E2 22026.528} C_VEL
LIN {X 0,Y 149.88,Z 526.81,A -85,B 0,C 180,E1 22038.33,E2 22038.33} C_VEL
LIN {X 0,Y 150.954,Z 526.81,A -85,B 0,C 180,E1 22047.181,E2 22047.181} C_VEL
LIN {X 0,Y 148.546,Z 526.81,A -85,B 0,C 180,E1 22050.379,E2 22050.379} C_VEL
LIN {X 0,Y 142.701,Z 526.81,A -85,B 0,C 180,E1 22055.851,E2 22055.851} C_VEL
LIN {X 0,Y 141.35,Z 526.81,A -85,B 0,C 180,E1 22065.353,E2 22065.353} C_VEL
LIN {X 0,Y 140.275,Z 526.81,A -85,B 0,C 180,E1 22075.562,E2 22075.562} C_VEL
LIN {X 0,Y 139.794,Z 526.81,A -85,B 0,C 180,E1 22082.771,E2 22082.771} C_VEL
LIN {X 0,Y 139.434,Z 526.81,A -85,B 0,C 180,E1 22090.637,E2 22090.637} C_VEL
LIN {X 0,Y 139.433,Z 526.81,A -85,B 0,C 180,E1 22099.451,E2 22099.451} C_VEL
LIN {X 0,Y 139.938,Z 526.81,A -85,B 0,C 180,E1 22109.918,E2 22109.918} C_VEL
LIN {X 0,Y 141.008,Z 526.81,A -85,B 0,C 180,E1 22121.19,E2 22121.19} C_VEL
LIN {X 0,Y 142.656,Z 526.81,A -85,B 0,C 180,E1 22133.889,E2 22133.889} C_VEL
LIN {X 0,Y 143.644,Z 526.81,A -85,B 0,C 180,E1 22139.981,E2 22139.981} C_VEL
LIN {X 0,Y 141.774,Z 526.81,A -85,B 0,C 180,E1 22152.313,E2 22152.313} C_VEL
LIN {X 0,Y 141.014,Z 526.81,A -85,B 0,C 180,E1 22158.769,E2 22158.769} C_VEL
LIN {X 0,Y 140.038,Z 526.81,A -85,B 0,C 180,E1 22170.153,E2 22170.153} C_VEL
LIN {X 0,Y 140.168,Z 527.607,A -85,B 0,C 180,E1 22181.733,E2 22181.733} C_VEL
LIN {X 0,Y 155.08,Z 585.392,A -85,B 0,C 180,E1 22188.344,E2 22188.344} C_VEL
LIN {X 0,Y 161.453,Z 611.786,A -85,B 0,C 180,E1 22192.404,E2 22192.404} C_VEL
LIN {X 0,Y 155.883,Z 641.554,A -85,B 0,C 180,E1 22198.545,E2 22198.545} C_VEL
LIN {X 0,Y 151.483,Z 666.805,A -85,B 0,C 180,E1 22206.449,E2 22206.449} C_VEL
LIN {X 0,Y 149.541,Z 688.206,A -85,B 0,C 180,E1 22216.412,E2 22216.412} C_VEL
LIN {X 0,Y 150.523,Z 701.578,A -85,B 0,C 180,E1 22225.687,E2 22225.687} C_VEL
LIN {X 0,Y 150.972,Z 705.796,A -85,B 0,C 180,E1 22230.014,E2 22230.014} C_VEL
LIN {X 0,Y 147.597,Z 710.412,A -85,B 0,C 180,E1 22241.853,E2 22241.853} C_VEL
LIN {X 0,Y 149.326,Z 710.682,A -85,B 0,C 180,E1 22254.191,E2 22254.191} C_VEL
LIN {X 0,Y 164.419,Z 705.495,A -85,B 0,C 180,E1 22270.152,E2 22270.152} C_VEL
LIN {X 0,Y 189.637,Z 695.594,A -85,B 0,C 180,E1 22281.135,E2 22281.135} C_VEL
LIN {X 0,Y 193.568,Z 693.952,A -85,B 0,C 180,E1 22282.279,E2 22282.279} C_VEL
LIN {X 0,Y 194.117,Z 693.411,A -85,B 0,C 180,E1 22282.957,E2 22282.957} C_VEL
LIN {X 0,Y 172.232,Z 692.506,A -85,B 0,C 180,E1 22291.557,E2 22291.557} C_VEL
LIN {X 0,Y 157.355,Z 685.578,A -85,B 0,C 180,E1 22301.796,E2 22301.796} C_VEL
LIN {X 0,Y 149.546,Z 673.275,A -85,B 0,C 180,E1 22312.748,E2 22312.748} C_VEL
LIN {X 0,Y 147.178,Z 655.183,A -85,B 0,C 180,E1 22323.704,E2 22323.704} C_VEL
LIN {X 0,Y 148.425,Z 631.64,A -85,B 0,C 180,E1 22333.455,E2 22333.455} C_VEL
LIN {X 0,Y 151.726,Z 603.982,A -85,B 0,C 180,E1 22341.225,E2 22341.225} C_VEL
LIN {X 0,Y 153.185,Z 587.734,A -85,B 0,C 180,E1 22344.572,E2 22344.572} C_VEL
LIN {X 0,Y 147.056,Z 555.987,A -85,B 0,C 180,E1 22349.881,E2 22349.881} C_VEL
LIN {X 0,Y 140.251,Z 526.81,A -85,B 0,C 180,E1 22353.894,E2 22353.894} C_VEL
LIN {X 0,Y 139.526,Z 526.81,A -85,B 0,C 180,E1 22360.647,E2 22360.647} C_VEL
LIN {X 0,Y 139.484,Z 526.81,A -85,B 0,C 180,E1 22369.476,E2 22369.476} C_VEL
LIN {X 0,Y 139.976,Z 526.81,A -85,B 0,C 180,E1 22379.953,E2 22379.953} C_VEL
LIN {X 0,Y 141.031,Z 526.81,A -85,B 0,C 180,E1 22391.196,E2 22391.196} C_VEL
LIN {X 0,Y 142.672,Z 526.81,A -85,B 0,C 180,E1 22403.894,E2 22403.894} C_VEL
LIN {X 0,Y 143.651,Z 526.81,A -85,B 0,C 180,E1 22409.986,E2 22409.986} C_VEL
LIN {X 0,Y 142.701,Z 526.81,A -85,B 0,C 180,E1 22415.851,E2 22415.851} C_VEL
LIN {X 0,Y 139.497,Z 526.81,A -85,B 0,C 180,E1 22420.984,E2 22420.984} C_VEL
LIN {X 0,Y 132.837,Z 526.81,A -85,B 0,C 180,E1 22429.977,E2 22429.977} C_VEL
LIN {X 0,Y 132.18,Z 526.81,A -85,B 0,C 180,E1 22437.252,E2 22437.252} C_VEL
LIN {X 0,Y 131.422,Z 526.81,A -85,B 0,C 180,E1 22446.219,E2 22446.219} C_VEL
LIN {X 0,Y 131.161,Z 526.81,A -85,B 0,C 180,E1 22456.137,E2 22456.137} C_VEL
LIN {X 0,Y 131.499,Z 526.81,A -85,B 0,C 180,E1 22464.829,E2 22464.829} C_VEL
LIN {X 0,Y 132.371,Z 526.81,A -85,B 0,C 180,E1 22476.174,E2 22476.174} C_VEL
LIN {X 0,Y 133.698,Z 526.81,A -85,B 0,C 180,E1 22486.89,E2 22486.89} C_VEL
LIN {X 0,Y 135.689,Z 526.81,A -85,B 0,C 180,E1 22499.98,E2 22499.98} C_VEL
LIN {X 0,Y 133.7,Z 526.81,A -85,B 0,C 180,E1 22513.069,E2 22513.069} C_VEL
LIN {X 0,Y 132.388,Z 526.81,A -85,B 0,C 180,E1 22523.843,E2 22523.843} C_VEL
LIN {X 0,Y 131.961,Z 526.81,A -85,B 0,C 180,E1 22539.708,E2 22539.708} C_VEL
LIN {X 0,Y 132.128,Z 526.81,A -85,B 0,C 180,E1 22540.799,E2 22540.799} C_VEL
LIN {X 0,Y 146.723,Z 584.748,A -85,B 0,C 180,E1 22547.845,E2 22547.845} C_VEL
LIN {X 0,Y 153.477,Z 612.045,A -85,B 0,C 180,E1 22552.293,E2 22552.293} C_VEL
LIN {X 0,Y 147.825,Z 641.44,A -85,B 0,C 180,E1 22558.783,E2 22558.783} C_VEL
LIN {X 0,Y 143.484,Z 667.309,A -85,B 0,C 180,E1 22567.526,E2 22567.526} C_VEL
LIN {X 0,Y 142.046,Z 687.526,A -85,B 0,C 180,E1 22577.706,E2 22577.706} C_VEL
LIN {X 0,Y 143.249,Z 700.016,A -85,B 0,C 180,E1 22586.985,E2 22586.985} C_VEL
LIN {X 0,Y 143.562,Z 702.905,A -85,B 0,C 180,E1 22590.014,E2 22590.014} C_VEL
LIN {X 0,Y 140.049,Z 707.902,A -85,B 0,C 180,E1 22602.502,E2 22602.502} C_VEL
LIN {X 0,Y 145.728,Z 707.857,A -85,B 0,C 180,E1 22621.314,E2 22621.314} C_VEL
LIN {X 0,Y 162.541,Z 703.034,A -85,B 0,C 180,E1 22634.334,E2 22634.334} C_VEL
LIN {X 0,Y 181.89,Z 696.494,A -85,B 0,C 180,E1 22642.181,E2 22642.181} C_VEL
LIN {X 0,Y 183.269,Z 695.758,A -85,B 0,C 180,E1 22643.034,E2 22643.034} C_VEL
LIN {X 0,Y 161.857,Z 692.569,A -85,B 0,C 180,E1 22652.134,E2 22652.134} C_VEL
LIN {X 0,Y 148.471,Z 684.43,A -85,B 0,C 180,E1 22662.206,E2 22662.206} C_VEL
LIN {X 0,Y 141.13,Z 670.463,A -85,B 0,C 180,E1 22673.861,E2 22673.861} C_VEL
LIN {X 0,Y 139.322,Z 651.986,A -85,B 0,C 180,E1 22684.694,E2 22684.694} C_VEL
LIN {X 0,Y 140.826,Z 628.586,A -85,B 0,C 180,E1 22694.295,E2 22694.295} C_VEL
LIN {X 0,Y 144.382,Z 599.697,A -85,B 0,C 180,E1 22702.361,E2 22702.361} C_VEL
LIN {X 0,Y 145.14,Z 587.241,A -85,B 0,C 180,E1 22704.982,E2 22704.982} C_VEL
LIN {X 0,Y 138.629,Z 554.267,A -85,B 0,C 180,E1 22710.691,E2 22710.691} C_VEL
LIN {X 0,Y 132.177,Z 526.81,A -85,B 0,C 180,E1 22714.537,E2 22714.537} C_VEL
LIN {X 0,Y 131.224,Z 526.81,A -85,B 0,C 180,E1 22726.167,E2 22726.167} C_VEL
LIN {X 0,Y 131.544,Z 526.81,A -85,B 0,C 180,E1 22734.846,E2 22734.846} C_VEL
LIN {X 0,Y 132.407,Z 526.81,A -85,B 0,C 180,E1 22746.22,E2 22746.22} C_VEL
LIN {X 0,Y 133.713,Z 526.81,A -85,B 0,C 180,E1 22756.895,E2 22756.895} C_VEL
LIN {X 0,Y 134.642,Z 526.81,A -85,B 0,C 180,E1 22763.528,E2 22763.528} C_VEL
LIN {X 0,Y 135.708,Z 526.81,A -85,B 0,C 180,E1 22769.985,E2 22769.985} C_VEL
LIN {X 0,Y 134.664,Z 526.81,A -85,B 0,C 180,E1 22776.44,E2 22776.44} C_VEL
LIN {X 0,Y 133.743,Z 526.81,A -85,B 0,C 180,E1 22783.07,E2 22783.07} C_VEL
LIN {X 0,Y 132.837,Z 526.81,A -85,B 0,C 180,E1 22789.977,E2 22789.977} C_VEL
LIN {X 0,Y 129.847,Z 526.81,A -85,B 0,C 180,E1 22795.52,E2 22795.52} C_VEL
LIN {X 0,Y 123.224,Z 526.81,A -85,B 0,C 180,E1 22805.267,E2 22805.267} C_VEL
LIN {X 0,Y 123.147,Z 526.81,A -85,B 0,C 180,E1 22817.51,E2 22817.51} C_VEL
LIN {X 0,Y 123.833,Z 526.81,A -85,B 0,C 180,E1 22830.698,E2 22830.698} C_VEL
LIN {X 0,Y 124.685,Z 526.81,A -85,B 0,C 180,E1 22838.614,E2 22838.614} C_VEL
LIN {X 0,Y 125.538,Z 526.81,A -85,B 0,C 180,E1 22846.021,E2 22846.021} C_VEL
LIN {X 0,Y 126.585,Z 526.81,A -85,B 0,C 180,E1 22853.608,E2 22853.608} C_VEL
LIN {X 0,Y 127.726,Z 526.81,A -85,B 0,C 180,E1 22859.979,E2 22859.979} C_VEL
LIN {X 0,Y 126.562,Z 526.81,A -85,B 0,C 180,E1 22866.849,E2 22866.849} C_VEL
LIN {X 0,Y 125.344,Z 526.81,A -85,B 0,C 180,E1 22874.971,E2 22874.971} C_VEL
LIN {X 0,Y 124.698,Z 526.81,A -85,B 0,C 180,E1 22881.338,E2 22881.338} C_VEL
LIN {X 0,Y 123.785,Z 526.81,A -85,B 0,C 180,E1 22891.14,E2 22891.14} C_VEL
LIN {X 0,Y 124.121,Z 527.492,A -85,B 0,C 180,E1 22900.024,E2 22900.024} C_VEL
LIN {X 0,Y 138.319,Z 583.882,A -85,B 0,C 180,E1 22907.313,E2 22907.313} C_VEL
LIN {X 0,Y 145.379,Z 612.701,A -85,B 0,C 180,E1 22912.294,E2 22912.294} C_VEL
LIN {X 0,Y 139.508,Z 642.82,A -85,B 0,C 180,E1 22919.543,E2 22919.543} C_VEL
LIN {X 0,Y 135.529,Z 667.57,A -85,B 0,C 180,E1 22928.727,E2 22928.727} C_VEL
LIN {X 0,Y 134.691,Z 687.237,A -85,B 0,C 180,E1 22939.49,E2 22939.49} C_VEL
LIN {X 0,Y 136.018,Z 698.343,A -85,B 0,C 180,E1 22948.42,E2 22948.42} C_VEL
LIN {X 0,Y 135.095,Z 701.713,A -85,B 0,C 180,E1 22953.228,E2 22953.228} C_VEL
LIN {X 0,Y 132.891,Z 706.207,A -85,B 0,C 180,E1 22970.003,E2 22970.003} C_VEL
LIN {X 0,Y 144.963,Z 704.638,A -85,B 0,C 180,E1 22988.823,E2 22988.823} C_VEL
LIN {X 0,Y 171.773,Z 697.677,A -85,B 0,C 180,E1 23002.514,E2 23002.514} C_VEL
LIN {X 0,Y 159.803,Z 694.936,A -85,B 0,C 180,E1 23008.297,E2 23008.297} C_VEL
LIN {X 0,Y 143.986,Z 687.09,A -85,B 0,C 180,E1 23018.426,E2 23018.426} C_VEL
LIN {X 0,Y 134.667,Z 673.785,A -85,B 0,C 180,E1 23030.312,E2 23030.312} C_VEL
LIN {X 0,Y 131.548,Z 654.83,A -85,B 0,C 180,E1 23042.494,E2 23042.494} C_VEL
LIN {X 0,Y 132.654,Z 630.867,A -85,B 0,C 180,E1 23053.215,E2 23053.215} C_VEL
LIN {X 0,Y 135.998,Z 603.247,A -85,B 0,C 180,E1 23061.66,E2 23061.66} C_VEL
LIN {X 0,Y 137.269,Z 588.085,A -85,B 0,C 180,E1 23065.105,E2 23065.105} C_VEL
LIN {X 0,Y 130.948,Z 555.976,A -85,B 0,C 180,E1 23071.001,E2 23071.001} C_VEL
LIN {X 0,Y 124.085,Z 526.81,A -85,B 0,C 180,E1 23075.492,E2 23075.492} C_VEL
LIN {X 0,Y 123.206,Z 526.81,A -85,B 0,C 180,E1 23087.534,E2 23087.534} C_VEL
LIN {X 0,Y 123.859,Z 526.81,A -85,B 0,C 180,E1 23100.708,E2 23100.708} C_VEL
LIN {X 0,Y 124.717,Z 526.81,A -85,B 0,C 180,E1 23108.624,E2 23108.624} C_VEL
LIN {X 0,Y 125.555,Z 526.81,A -85,B 0,C 180,E1 23116.027,E2 23116.027} C_VEL
LIN {X 0,Y 126.583,Z 526.81,A -85,B 0,C 180,E1 23123.114,E2 23123.114} C_VEL
LIN {X 0,Y 127.745,Z 526.81,A -85,B 0,C 180,E1 23129.984,E2 23129.984} C_VEL
LIN {X 0,Y 126.607,Z 526.81,A -85,B 0,C 180,E1 23136.852,E2 23136.852} C_VEL
LIN {X 0,Y 125.393,Z 526.81,A -85,B 0,C 180,E1 23144.92,E2 23144.92} C_VEL
LIN {X 0,Y 124.719,Z 526.81,A -85,B 0,C 180,E1 23151.34,E2 23151.34} C_VEL
LIN {X 0,Y 123.674,Z 526.81,A -85,B 0,C 180,E1 23160.985,E2 23160.985} C_VEL
LIN {X 0,Y 123.224,Z 526.81,A -85,B 0,C 180,E1 23165.267,E2 23165.267} C_VEL
LIN {X 0,Y 120.527,Z 526.81,A -85,B 0,C 180,E1 23171.264,E2 23171.264} C_VEL
LIN {X 0,Y 115.354,Z 526.81,A -85,B 0,C 180,E1 23181.803,E2 23181.803} C_VEL
LIN {X 0,Y 116.193,Z 526.81,A -85,B 0,C 180,E1 23195.76,E2 23195.76} C_VEL
LIN {X 0,Y 117.412,Z 526.81,A -85,B 0,C 180,E1 23205.031,E2 23205.031} C_VEL
LIN {X 0,Y 118.546,Z 526.81,A -85,B 0,C 180,E1 23213.751,E2 23213.751} C_VEL
LIN {X 0,Y 119.763,Z 526.81,A -85,B 0,C 180,E1 23219.978,E2 23219.978} C_VEL
LIN {X 0,Y 118.479,Z 526.81,A -85,B 0,C 180,E1 23227.319,E2 23227.319} C_VEL
LIN {X 0,Y 117.417,Z 526.81,A -85,B 0,C 180,E1 23234.921,E2 23234.921} C_VEL
LIN {X 0,Y 116.227,Z 526.81,A -85,B 0,C 180,E1 23244.277,E2 23244.277} C_VEL
LIN {X 0,Y 116.075,Z 526.81,A -85,B 0,C 180,E1 23258.963,E2 23258.963} C_VEL
LIN {X 0,Y 130.031,Z 583.438,A -85,B 0,C 180,E1 23266.846,E2 23266.846} C_VEL
LIN {X 0,Y 137.428,Z 612.477,A -85,B 0,C 180,E1 23272.176,E2 23272.176} C_VEL
LIN {X 0,Y 131.796,Z 641.17,A -85,B 0,C 180,E1 23279.519,E2 23279.519} C_VEL
LIN {X 0,Y 127.883,Z 665.911,A -85,B 0,C 180,E1 23289.212,E2 23289.212} C_VEL
LIN {X 0,Y 127.349,Z 685.595,A -85,B 0,C 180,E1 23300.608,E2 23300.608} C_VEL
LIN {X 0,Y 128.853,Z 696.533,A -85,B 0,C 180,E1 23310.016,E2 23310.016} C_VEL
LIN {X 0,Y 125.632,Z 701.361,A -85,B 0,C 180,E1 23320.431,E2 23320.431} C_VEL
LIN {X 0,Y 128.074,Z 703.919,A -85,B 0,C 180,E1 23338.239,E2 23338.239} C_VEL
LIN {X 0,Y 146.987,Z 701.325,A -85,B 0,C 180,E1 23356.161,E2 23356.161} C_VEL
LIN {X 0,Y 160.31,Z 698.407,A -85,B 0,C 180,E1 23362.303,E2 23362.303} C_VEL
LIN {X 0,Y 159.87,Z 697.672,A -85,B 0,C 180,E1 23363.594,E2 23363.594} C_VEL
LIN {X 0,Y 140.172,Z 689.606,A -85,B 0,C 180,E1 23374.424,E2 23374.424} C_VEL
LIN {X 0,Y 128.277,Z 675.941,A -85,B 0,C 180,E1 23387.236,E2 23387.236} C_VEL
LIN {X 0,Y 123.941,Z 657.463,A -85,B 0,C 180,E1 23400.022,E2 23400.022} C_VEL
LIN {X 0,Y 124.437,Z 634.423,A -85,B 0,C 180,E1 23411.425,E2 23411.425} C_VEL
LIN {X 0,Y 127.601,Z 606.529,A -85,B 0,C 180,E1 23420.874,E2 23420.874} C_VEL
LIN {X 0,Y 129.335,Z 588.427,A -85,B 0,C 180,E1 23425.308,E2 23425.308} C_VEL
LIN {X 0,Y 122.77,Z 555.431,A -85,B 0,C 180,E1 23431.686,E2 23431.686} C_VEL
LIN {X 0,Y 116,Z 526.81,A -85,B 0,C 180,E1 23436.389,E2 23436.389} C_VEL
LIN {X 0,Y 115.418,Z 526.81,A -85,B 0,C 180,E1 23451.948,E2 23451.948} C_VEL
LIN {X 0,Y 116.229,Z 526.81,A -85,B 0,C 180,E1 23465.813,E2 23465.813} C_VEL
LIN {X 0,Y 117.433,Z 526.81,A -85,B 0,C 180,E1 23475.039,E2 23475.039} C_VEL
LIN {X 0,Y 118.498,Z 526.81,A -85,B 0,C 180,E1 23482.642,E2 23482.642} C_VEL
LIN {X 0,Y 119.792,Z 526.81,A -85,B 0,C 180,E1 23489.983,E2 23489.983} C_VEL
LIN {X 0,Y 118.523,Z 526.81,A -85,B 0,C 180,E1 23497.322,E2 23497.322} C_VEL
LIN {X 0,Y 117.455,Z 526.81,A -85,B 0,C 180,E1 23504.922,E2 23504.922} C_VEL
LIN {X 0,Y 116.223,Z 526.81,A -85,B 0,C 180,E1 23514.18,E2 23514.18} C_VEL
LIN {X 0,Y 115.375,Z 526.81,A -85,B 0,C 180,E1 23528.025,E2 23528.025} C_VEL
LIN {X 0,Y 115.354,Z 526.81,A -85,B 0,C 180,E1 23541.803,E2 23541.803} C_VEL
LIN {X 0,Y 113.181,Z 526.81,A -85,B 0,C 180,E1 23548.24,E2 23548.24} C_VEL
LIN {X 0,Y 108.365,Z 526.81,A -85,B 0,C 180,E1 23559.583,E2 23559.583} C_VEL
LIN {X 0,Y 109.515,Z 526.81,A -85,B 0,C 180,E1 23565.337,E2 23565.337} C_VEL
LIN {X 0,Y 111.776,Z 526.81,A -85,B 0,C 180,E1 23579.976,E2 23579.976} C_VEL
LIN {X 0,Y 109.516,Z 526.81,A -85,B 0,C 180,E1 23594.664,E2 23594.664} C_VEL
LIN {X 0,Y 108.223,Z 526.81,A -85,B 0,C 180,E1 23604.787,E2 23604.787} C_VEL
LIN {X 0,Y 108.068,Z 526.81,A -85,B 0,C 180,E1 23617.983,E2 23617.983} C_VEL
LIN {X 0,Y 121.93,Z 583.565,A -85,B 0,C 180,E1 23626.488,E2 23626.488} C_VEL
LIN {X 0,Y 129.333,Z 613.081,A -85,B 0,C 180,E1 23632.277,E2 23632.277} C_VEL
LIN {X 0,Y 123.498,Z 642.653,A -85,B 0,C 180,E1 23640.653,E2 23640.653} C_VEL
LIN {X 0,Y 120.11,Z 666.026,A -85,B 0,C 180,E1 23650.77,E2 23650.77} C_VEL
LIN {X 0,Y 120.171,Z 684.988,A -85,B 0,C 180,E1 23662.779,E2 23662.779} C_VEL
LIN {X 0,Y 121.513,Z 693.036,A -85,B 0,C 180,E1 23670.017,E2 23670.017} C_VEL
LIN {X 0,Y 118.439,Z 698.106,A -85,B 0,C 180,E1 23680.684,E2 23680.684} C_VEL
LIN {X 0,Y 121.336,Z 701.309,A -85,B 0,C 180,E1 23699.962,E2 23699.962} C_VEL
LIN {X 0,Y 141.669,Z 699.512,A -85,B 0,C 180,E1 23718.449,E2 23718.449} C_VEL
LIN {X 0,Y 151.141,Z 697.804,A -85,B 0,C 180,E1 23723.079,E2 23723.079} C_VEL
LIN {X 0,Y 131.229,Z 688.137,A -85,B 0,C 180,E1 23734.388,E2 23734.388} C_VEL
LIN {X 0,Y 119.676,Z 672.672,A -85,B 0,C 180,E1 23748.16,E2 23748.16} C_VEL
LIN {X 0,Y 116.027,Z 652.324,A -85,B 0,C 180,E1 23761.892,E2 23761.892} C_VEL
LIN {X 0,Y 117.136,Z 627.621,A -85,B 0,C 180,E1 23773.655,E2 23773.655} C_VEL
LIN {X 0,Y 120.777,Z 598.538,A -85,B 0,C 180,E1 23783.073,E2 23783.073} C_VEL
LIN {X 0,Y 121.173,Z 587.354,A -85,B 0,C 180,E1 23785.81,E2 23785.81} C_VEL
LIN {X 0,Y 114.34,Z 553.598,A -85,B 0,C 180,E1 23792.609,E2 23792.609} C_VEL
LIN {X 0,Y 107.927,Z 526.81,A -85,B 0,C 180,E1 23797.121,E2 23797.121} C_VEL
LIN {X 0,Y 107.188,Z 526.81,A -85,B 0,C 180,E1 23805.041,E2 23805.041} C_VEL
LIN {X 0,Y 107.647,Z 526.81,A -85,B 0,C 180,E1 23817.597,E2 23817.597} C_VEL
LIN {X 0,Y 108.182,Z 526.81,A -85,B 0,C 180,E1 23825.153,E2 23825.153} C_VEL
LIN {X 0,Y 109.538,Z 526.81,A -85,B 0,C 180,E1 23835.452,E2 23835.452} C_VEL
LIN {X 0,Y 111.804,Z 526.81,A -85,B 0,C 180,E1 23849.982,E2 23849.982} C_VEL
LIN {X 0,Y 109.566,Z 526.81,A -85,B 0,C 180,E1 23864.604,E2 23864.604} C_VEL
LIN {X 0,Y 108.179,Z 526.81,A -85,B 0,C 180,E1 23874.806,E2 23874.806} C_VEL
LIN {X 0,Y 107.473,Z 526.81,A -85,B 0,C 180,E1 23884.276,E2 23884.276} C_VEL
LIN {X 0,Y 107.066,Z 526.81,A -85,B 0,C 180,E1 23894.97,E2 23894.97} C_VEL
LIN {X 0,Y 107.607,Z 526.81,A -85,B 0,C 180,E1 23907.553,E2 23907.553} C_VEL
LIN {X 0,Y 108.365,Z 526.81,A -85,B 0,C 180,E1 23919.583,E2 23919.583} C_VEL
LIN {X 0,Y 106.65,Z 526.81,A -85,B 0,C 180,E1 23926.513,E2 23926.513} C_VEL
LIN {X 0,Y 103.401,Z 526.81,A -85,B 0,C 180,E1 23938.653,E2 23938.653} C_VEL
LIN {X 0,Y 102.301,Z 526.81,A -85,B 0,C 180,E1 23948.484,E2 23948.484} C_VEL
LIN {X 0,Y 100.256,Z 526.81,A -85,B 0,C 180,E1 23965.074,E2 23965.074} C_VEL
LIN {X 0,Y 100.07,Z 526.81,A -85,B 0,C 180,E1 23976.959,E2 23976.959} C_VEL
LIN {X 0,Y 113.673,Z 583.025,A -85,B 0,C 180,E1 23986.025,E2 23986.025} C_VEL
LIN {X 0,Y 121.405,Z 612.923,A -85,B 0,C 180,E1 23992.288,E2 23992.288} C_VEL
LIN {X 0,Y 115.656,Z 641.858,A -85,B 0,C 180,E1 24001.156,E2 24001.156} C_VEL
LIN {X 0,Y 112.475,Z 665.341,A -85,B 0,C 180,E1 24012.174,E2 24012.174} C_VEL
LIN {X 0,Y 113.21,Z 684.11,A -85,B 0,C 180,E1 24025.085,E2 24025.085} C_VEL
LIN {X 0,Y 114.049,Z 690.921,A -85,B 0,C 180,E1 24032.039,E2 24032.039} C_VEL
LIN {X 0,Y 110.777,Z 696.36,A -85,B 0,C 180,E1 24047.008,E2 24047.008} C_VEL
LIN {X 0,Y 120.165,Z 698.722,A -85,B 0,C 180,E1 24069.072,E2 24069.072} C_VEL
LIN {X 0,Y 138.525,Z 697.202,A -85,B 0,C 180,E1 24081.902,E2 24081.902} C_VEL
LIN {X 0,Y 139.681,Z 696.505,A -85,B 0,C 180,E1 24083.451,E2 24083.451} C_VEL
LIN {X 0,Y 120.508,Z 684.409,A -85,B 0,C 180,E1 24095.925,E2 24095.925} C_VEL
LIN {X 0,Y 110.737,Z 667.621,A -85,B 0,C 180,E1 24110.184,E2 24110.184} C_VEL
LIN {X 0,Y 108.2,Z 646.326,A -85,B 0,C 180,E1 24124.037,E2 24124.037} C_VEL
LIN {X 0,Y 110.068,Z 620.464,A -85,B 0,C 180,E1 24135.993,E2 24135.993} C_VEL
LIN {X 0,Y 113.816,Z 591.431,A -85,B 0,C 180,E1 24145.013,E2 24145.013} C_VEL
LIN {X 0,Y 107.46,Z 559.082,A -85,B 0,C 180,E1 24152.252,E2 24152.252} C_VEL
LIN {X 0,Y 99.854,Z 526.81,A -85,B 0,C 180,E1 24158.354,E2 24158.354} C_VEL
LIN {X 0,Y 99.092,Z 526.81,A -85,B 0,C 180,E1 24172.299,E2 24172.299} C_VEL
LIN {X 0,Y 100.233,Z 526.81,A -85,B 0,C 180,E1 24185.059,E2 24185.059} C_VEL
LIN {X 0,Y 102.322,Z 526.81,A -85,B 0,C 180,E1 24201.47,E2 24201.47} C_VEL
LIN {X 0,Y 103.818,Z 526.81,A -85,B 0,C 180,E1 24209.98,E2 24209.98} C_VEL
LIN {X 0,Y 102.347,Z 526.81,A -85,B 0,C 180,E1 24218.487,E2 24218.487} C_VEL
LIN {X 0,Y 100.954,Z 526.81,A -85,B 0,C 180,E1 24227.433,E2 24227.433} C_VEL
LIN {X 0,Y 99.916,Z 526.81,A -85,B 0,C 180,E1 24237.016,E2 24237.016} C_VEL
LIN {X 0,Y 98.89,Z 526.81,A -85,B 0,C 180,E1 24250.008,E2 24250.008} C_VEL
LIN {X 0,Y 99.017,Z 526.81,A -85,B 0,C 180,E1 24262.26,E2 24262.26} C_VEL
LIN {X 0,Y 100.191,Z 526.81,A -85,B 0,C 180,E1 24275.006,E2 24275.006} C_VEL
LIN {X 0,Y 100.913,Z 526.81,A -85,B 0,C 180,E1 24282.511,E2 24282.511} C_VEL
LIN {X 0,Y 102.533,Z 526.81,A -85,B 0,C 180,E1 24294.261,E2 24294.261} C_VEL
LIN {X 0,Y 103.401,Z 526.81,A -85,B 0,C 180,E1 24298.653,E2 24298.653} C_VEL
LIN {X 0,Y 102.055,Z 526.81,A -85,B 0,C 180,E1 24303.944,E2 24303.944} C_VEL
LIN {X 0,Y 92.734,Z 526.81,A -85,B 0,C 180,E1 24318.518,E2 24318.518} C_VEL
LIN {X 0,Y 92.13,Z 527.486,A -85,B 0,C 180,E1 24335.973,E2 24335.973} C_VEL
LIN {X 0,Y 105.329,Z 582.365,A -85,B 0,C 180,E1 24345.542,E2 24345.542} C_VEL
LIN {X 0,Y 113.278,Z 613.426,A -85,B 0,C 180,E1 24352.557,E2 24352.557} C_VEL
LIN {X 0,Y 107.625,Z 642.096,A -85,B 0,C 180,E1 24362.247,E2 24362.247} C_VEL
LIN {X 0,Y 104.966,Z 665.411,A -85,B 0,C 180,E1 24374.329,E2 24374.329} C_VEL
LIN {X 0,Y 106.404,Z 682.968,A -85,B 0,C 180,E1 24387.572,E2 24387.572} C_VEL
LIN {X 0,Y 106.789,Z 687.535,A -85,B 0,C 180,E1 24392.788,E2 24392.788} C_VEL
LIN {X 0,Y 103.755,Z 692.711,A -85,B 0,C 180,E1 24406.99,E2 24406.99} C_VEL
LIN {X 0,Y 114.353,Z 695.911,A -85,B 0,C 180,E1 24431.478,E2 24431.478} C_VEL
LIN {X 0,Y 128.178,Z 695.501,A -85,B 0,C 180,E1 24441.596,E2 24441.596} C_VEL
LIN {X 0,Y 129.632,Z 694.932,A -85,B 0,C 180,E1 24443.208,E2 24443.208} C_VEL
LIN {X 0,Y 111.642,Z 681.667,A -85,B 0,C 180,E1 24456.02,E2 24456.02} C_VEL
LIN {X 0,Y 102.368,Z 663.044,A -85,B 0,C 180,E1 24471.521,E2 24471.521} C_VEL
LIN {X 0,Y 100.486,Z 641.506,A -85,B 0,C 180,E1 24485.43,E2 24485.43} C_VEL
LIN {X 0,Y 102.701,Z 614.744,A -85,B 0,C 180,E1 24497.728,E2 24497.728} C_VEL
LIN {X 0,Y 105.692,Z 590.302,A -85,B 0,C 180,E1 24505.479,E2 24505.479} C_VEL
LIN {X 0,Y 98.837,Z 556.325,A -85,B 0,C 180,E1 24513.442,E2 24513.442} C_VEL
LIN {X 0,Y 91.851,Z 526.81,A -85,B 0,C 180,E1 24519.333,E2 24519.333} C_VEL
LIN {X 0,Y 91.099,Z 526.81,A -85,B 0,C 180,E1 24536.25,E2 24536.25} C_VEL
LIN {X 0,Y 92.716,Z 526.81,A -85,B 0,C 180,E1 24550.914,E2 24550.914} C_VEL
LIN {X 0,Y 94.116,Z 526.81,A -85,B 0,C 180,E1 24560.72,E2 24560.72} C_VEL
LIN {X 0,Y 95.801,Z 526.81,A -85,B 0,C 180,E1 24569.979,E2 24569.979} C_VEL
LIN {X 0,Y 93.368,Z 526.81,A -85,B 0,C 180,E1 24583.24,E2 24583.24} C_VEL
LIN {X 0,Y 92.727,Z 526.81,A -85,B 0,C 180,E1 24589.037,E2 24589.037} C_VEL
LIN {X 0,Y 91.053,Z 526.81,A -85,B 0,C 180,E1 24603.707,E2 24603.707} C_VEL
LIN {X 0,Y 90.751,Z 526.81,A -85,B 0,C 180,E1 24618.1,E2 24618.1} C_VEL
LIN {X 0,Y 91.395,Z 526.81,A -85,B 0,C 180,E1 24630.167,E2 24630.167} C_VEL
LIN {X 0,Y 92.687,Z 526.81,A -85,B 0,C 180,E1 24640.902,E2 24640.902} C_VEL
LIN {X 0,Y 94.505,Z 526.81,A -85,B 0,C 180,E1 24654.699,E2 24654.699} C_VEL
LIN {X 0,Y 95.769,Z 526.81,A -85,B 0,C 180,E1 24659.972,E2 24659.972} C_VEL
LIN {X 0,Y 93.334,Z 526.81,A -85,B 0,C 180,E1 24673.359,E2 24673.359} C_VEL
LIN {X 0,Y 92.734,Z 526.81,A -85,B 0,C 180,E1 24678.518,E2 24678.518} C_VEL
LIN {X 0,Y 89.837,Z 526.81,A -85,B 0,C 180,E1 24683.686,E2 24683.686} C_VEL
LIN {X 0,Y 84.017,Z 526.81,A -85,B 0,C 180,E1 24692.861,E2 24692.861} C_VEL
LIN {X 0,Y 84.174,Z 527.619,A -85,B 0,C 180,E1 24694.757,E2 24694.757} C_VEL
LIN {X 0,Y 96.965,Z 581.374,A -85,B 0,C 180,E1 24704.993,E2 24704.993} C_VEL
LIN {X 0,Y 105.346,Z 612.974,A -85,B 0,C 180,E1 24712.669,E2 24712.669} C_VEL
LIN {X 0,Y 99.744,Z 642.01,A -85,B 0,C 180,E1 24723.444,E2 24723.444} C_VEL
LIN {X 0,Y 97.637,Z 664.964,A -85,B 0,C 180,E1 24736.571,E2 24736.571} C_VEL
LIN {X 0,Y 99.683,Z 681.309,A -85,B 0,C 180,E1 24750.021,E2 24750.021} C_VEL
LIN {X 0,Y 99.267,Z 684.518,A -85,B 0,C 180,E1 24754.618,E2 24754.618} C_VEL
LIN {X 0,Y 98.292,Z 691.064,A -85,B 0,C 180,E1 24777.547,E2 24777.547} C_VEL
LIN {X 0,Y 118.782,Z 693.003,A -85,B 0,C 180,E1 24801.667,E2 24801.667} C_VEL
LIN {X 0,Y 120.214,Z 692.912,A -85,B 0,C 180,E1 24802.663,E2 24802.663} C_VEL
LIN {X 0,Y 102.157,Z 677.254,A -85,B 0,C 180,E1 24817.134,E2 24817.134} C_VEL
LIN {X 0,Y 93.786,Z 656.231,A -85,B 0,C 180,E1 24834.238,E2 24834.238} C_VEL
LIN {X 0,Y 93.107,Z 632.908,A -85,B 0,C 180,E1 24848.798,E2 24848.798} C_VEL
LIN {X 0,Y 96.194,Z 603.748,A -85,B 0,C 180,E1 24861.374,E2 24861.374} C_VEL
LIN {X 0,Y 97.54,Z 589.695,A -85,B 0,C 180,E1 24865.775,E2 24865.775} C_VEL
LIN {X 0,Y 90.877,Z 556.72,A -85,B 0,C 180,E1 24874.053,E2 24874.053} C_VEL
LIN {X 0,Y 83.754,Z 526.81,A -85,B 0,C 180,E1 24880.59,E2 24880.59} C_VEL
LIN {X 0,Y 83.231,Z 526.81,A -85,B 0,C 180,E1 24896.896,E2 24896.896} C_VEL
LIN {X 0,Y 84.261,Z 526.81,A -85,B 0,C 180,E1 24908.912,E2 24908.912} C_VEL
LIN {X 0,Y 85.938,Z 526.81,A -85,B 0,C 180,E1 24919.828,E2 24919.828} C_VEL
LIN {X 0,Y 87.776,Z 526.81,A -85,B 0,C 180,E1 24929.977,E2 24929.977} C_VEL
LIN {X 0,Y 85.958,Z 526.81,A -85,B 0,C 180,E1 24940.121,E2 24940.121} C_VEL
LIN {X 0,Y 83.695,Z 526.81,A -85,B 0,C 180,E1 24955.174,E2 24955.174} C_VEL
LIN {X 0,Y 83.187,Z 526.81,A -85,B 0,C 180,E1 24963.065,E2 24963.065} C_VEL
LIN {X 0,Y 82.776,Z 526.81,A -85,B 0,C 180,E1 24976.988,E2 24976.988} C_VEL
LIN {X 0,Y 83.168,Z 526.81,A -85,B 0,C 180,E1 24986.86,E2 24986.86} C_VEL
LIN {X 0,Y 84.226,Z 526.81,A -85,B 0,C 180,E1 24998.896,E2 24998.896} C_VEL
LIN {X 0,Y 85.912,Z 526.81,A -85,B 0,C 180,E1 25009.818,E2 25009.818} C_VEL
LIN {X 0,Y 87.741,Z 526.81,A -85,B 0,C 180,E1 25019.97,E2 25019.97} C_VEL
LIN {X 0,Y 85.924,Z 526.81,A -85,B 0,C 180,E1 25030.117,E2 25030.117} C_VEL
LIN {X 0,Y 83.989,Z 526.81,A -85,B 0,C 180,E1 25045.721,E2 25045.721} C_VEL
LIN {X 0,Y 84.017,Z 526.81,A -85,B 0,C 180,E1 25052.861,E2 25052.861} C_VEL
LIN {X 0,Y 85.633,Z 529.75,A -85,B 0,C 180,E1 25055.252,E2 25055.252} C_VEL
LIN {X 0,Y 83.367,Z 558.195,A -85,B 0,C 180,E1 25059.711,E2 25059.711} C_VEL
LIN {X 0,Y 83.747,Z 560.282,A -85,B 0,C 180,E1 25060.144,E2 25060.144} C_VEL
LIN {X 0,Y 92.692,Z 596.179,A -85,B 0,C 180,E1 25068.378,E2 25068.378} C_VEL
LIN {X 0,Y 97.064,Z 614.244,A -85,B 0,C 180,E1 25073.443,E2 25073.443} C_VEL
LIN {X 0,Y 91.932,Z 641.78,A -85,B 0,C 180,E1 25084.871,E2 25084.871} C_VEL
LIN {X 0,Y 90.488,Z 664.354,A -85,B 0,C 180,E1 25099.173,E2 25099.173} C_VEL
LIN {X 0,Y 92.898,Z 678.827,A -85,B 0,C 180,E1 25112.108,E2 25112.108} C_VEL
LIN {X 0,Y 90.293,Z 683.931,A -85,B 0,C 180,E1 25124.482,E2 25124.482} C_VEL
LIN {X 0,Y 96.518,Z 688.828,A -85,B 0,C 180,E1 25148.892,E2 25148.892} C_VEL
LIN {X 0,Y 110.09,Z 689.703,A -85,B 0,C 180,E1 25162.528,E2 25162.528} C_VEL
LIN {X 0,Y 92.737,Z 672.056,A -85,B 0,C 180,E1 25178.48,E2 25178.48} C_VEL
LIN {X 0,Y 85.775,Z 650.085,A -85,B 0,C 180,E1 25196.236,E2 25196.236} C_VEL
LIN {X 0,Y 85.85,Z 624.248,A -85,B 0,C 180,E1 25212.046,E2 25212.046} C_VEL
LIN {X 0,Y 89.719,Z 593.536,A -85,B 0,C 180,E1 25224.636,E2 25224.636} C_VEL
LIN {X 0,Y 84.51,Z 564.818,A -85,B 0,C 180,E1 25232.825,E2 25232.825} C_VEL
LIN {X 0,Y 75.635,Z 526.81,A -85,B 0,C 180,E1 25241.641,E2 25241.641} C_VEL
LIN {X 0,Y 75.028,Z 526.81,A -85,B 0,C 180,E1 25253.88,E2 25253.88} C_VEL
LIN {X 0,Y 75.984,Z 526.81,A -85,B 0,C 180,E1 25266.485,E2 25266.485} C_VEL
LIN {X 0,Y 77.595,Z 526.81,A -85,B 0,C 180,E1 25278.721,E2 25278.721} C_VEL
LIN {X 0,Y 79.704,Z 526.81,A -85,B 0,C 180,E1 25289.974,E2 25289.974} C_VEL
LIN {X 0,Y 77.445,Z 526.81,A -85,B 0,C 180,E1 25302.022,E2 25302.022} C_VEL
LIN {X 0,Y 75.976,Z 526.81,A -85,B 0,C 180,E1 25313.459,E2 25313.459} C_VEL
LIN {X 0,Y 74.802,Z 526.81,A -85,B 0,C 180,E1 25327.355,E2 25327.355} C_VEL
LIN {X 0,Y 74.883,Z 526.81,A -85,B 0,C 180,E1 25343.929,E2 25343.929} C_VEL
LIN {X 0,Y 75.94,Z 526.81,A -85,B 0,C 180,E1 25356.463,E2 25356.463} C_VEL
LIN {X 0,Y 77.567,Z 526.81,A -85,B 0,C 180,E1 25368.709,E2 25368.709} C_VEL
LIN {X 0,Y 79.669,Z 526.81,A -85,B 0,C 180,E1 25379.966,E2 25379.966} C_VEL
LIN {X 0,Y 77.41,Z 526.81,A -85,B 0,C 180,E1 25392.18,E2 25392.18} C_VEL
LIN {X 0,Y 76.154,Z 526.999,A -85,B 0,C 180,E1 25413.244,E2 25413.244} C_VEL
LIN {X 0,Y 83.747,Z 560.282,A -85,B 0,C 180,E1 25420.144,E2 25420.144} C_VEL
LIN {X 0,Y 84.499,Z 568.814,A -85,B 0,C 180,E1 25421.804,E2 25421.804} C_VEL
LIN {X 0,Y 83.447,Z 591.615,A -85,B 0,C 180,E1 25427.2,E2 25427.2} C_VEL
LIN {X 0,Y 83.831,Z 593.572,A -85,B 0,C 180,E1 25427.736,E2 25427.736} C_VEL
LIN {X 0,Y 89.11,Z 613.691,A -85,B 0,C 180,E1 25433.814,E2 25433.814} C_VEL
LIN {X 0,Y 84.16,Z 641.874,A -85,B 0,C 180,E1 25446.854,E2 25446.854} C_VEL
LIN {X 0,Y 83.681,Z 664.586,A -85,B 0,C 180,E1 25463.066,E2 25463.066} C_VEL
LIN {X 0,Y 85.959,Z 675.958,A -85,B 0,C 180,E1 25474.537,E2 25474.537} C_VEL
LIN {X 0,Y 84.09,Z 682.424,A -85,B 0,C 180,E1 25495.886,E2 25495.886} C_VEL
LIN {X 0,Y 99.778,Z 686.309,A -85,B 0,C 180,E1 25520.933,E2 25520.933} C_VEL
LIN {X 0,Y 99.67,Z 685.445,A -85,B 0,C 180,E1 25522.618,E2 25522.618} C_VEL
LIN {X 0,Y 83.414,Z 665.88,A -85,B 0,C 180,E1 25540.138,E2 25540.138} C_VEL
LIN {X 0,Y 77.888,Z 643.138,A -85,B 0,C 180,E1 25558.642,E2 25558.642} C_VEL
LIN {X 0,Y 78.867,Z 616.014,A -85,B 0,C 180,E1 25575.064,E2 25575.064} C_VEL
LIN {X 0,Y 81.791,Z 591.078,A -85,B 0,C 180,E1 25585.398,E2 25585.398} C_VEL
LIN {X 0,Y 75.12,Z 558.427,A -85,B 0,C 180,E1 25595.161,E2 25595.161} C_VEL
LIN {X 0,Y 67.463,Z 526.81,A -85,B 0,C 180,E1 25603.892,E2 25603.892} C_VEL
LIN {X 0,Y 67.541,Z 526.81,A -85,B 0,C 180,E1 25623.809,E2 25623.809} C_VEL
LIN {X 0,Y 69.261,Z 526.81,A -85,B 0,C 180,E1 25637.343,E2 25637.343} C_VEL
LIN {X 0,Y 71.584,Z 526.81,A -85,B 0,C 180,E1 25649.971,E2 25649.971} C_VEL
LIN {X 0,Y 69.275,Z 526.81,A -85,B 0,C 180,E1 25662.594,E2 25662.594} C_VEL
LIN {X 0,Y 67.396,Z 526.81,A -85,B 0,C 180,E1 25676.665,E2 25676.665} C_VEL
LIN {X 0,Y 66.268,Z 526.81,A -85,B 0,C 180,E1 25696.678,E2 25696.678} C_VEL
LIN {X 0,Y 67.472,Z 526.81,A -85,B 0,C 180,E1 25713.774,E2 25713.774} C_VEL
LIN {X 0,Y 69.23,Z 526.81,A -85,B 0,C 180,E1 25727.328,E2 25727.328} C_VEL
LIN {X 0,Y 71.55,Z 526.81,A -85,B 0,C 180,E1 25739.963,E2 25739.963} C_VEL
LIN {X 0,Y 69.316,Z 526.81,A -85,B 0,C 180,E1 25752.577,E2 25752.577} C_VEL
LIN {X 0,Y 68.117,Z 526.81,A -85,B 0,C 180,E1 25771.573,E2 25771.573} C_VEL
LIN {X 0,Y 80.269,Z 579.851,A -85,B 0,C 180,E1 25784.022,E2 25784.022} C_VEL
LIN {X 0,Y 83.831,Z 593.572,A -85,B 0,C 180,E1 25787.736,E2 25787.736} C_VEL
LIN {X 0,Y 83.46,Z 604.282,A -85,B 0,C 180,E1 25791.001,E2 25791.001} C_VEL
LIN {X 0,Y 80.821,Z 614.662,A -85,B 0,C 180,E1 25794.968,E2 25794.968} C_VEL
LIN {X 0,Y 76.481,Z 642.488,A -85,B 0,C 180,E1 25809.759,E2 25809.759} C_VEL
LIN {X 0,Y 77.403,Z 664.74,A -85,B 0,C 180,E1 25827.785,E2 25827.785} C_VEL
LIN {X 0,Y 79.159,Z 670.883,A -85,B 0,C 180,E1 25834.125,E2 25834.125} C_VEL
LIN {X 0,Y 77.18,Z 677.182,A -85,B 0,C 180,E1 25853.13,E2 25853.13} C_VEL
LIN {X 0,Y 90.637,Z 682.081,A -85,B 0,C 180,E1 25880.227,E2 25880.227} C_VEL
LIN {X 0,Y 90.367,Z 681.176,A -85,B 0,C 180,E1 25881.953,E2 25881.953} C_VEL
LIN {X 0,Y 74.935,Z 660.337,A -85,B 0,C 180,E1 25900.871,E2 25900.871} C_VEL
LIN {X 0,Y 70.114,Z 636.269,A -85,B 0,C 180,E1 25920.811,E2 25920.811} C_VEL
LIN {X 0,Y 71.771,Z 608.253,A -85,B 0,C 180,E1 25937.815,E2 25937.815} C_VEL
LIN {X 0,Y 73.827,Z 591.145,A -85,B 0,C 180,E1 25945.221,E2 25945.221} C_VEL
LIN {X 0,Y 67.196,Z 558.965,A -85,B 0,C 180,E1 25955.844,E2 25955.844} C_VEL
LIN {X 0,Y 59.446,Z 526.81,A -85,B 0,C 180,E1 25965.785,E2 25965.785} C_VEL
LIN {X 0,Y 58.987,Z 526.81,A -85,B 0,C 180,E1 25979.072,E2 25979.072} C_VEL
LIN {X 0,Y 61.555,Z 526.81,A -85,B 0,C 180,E1 25999.929,E2 25999.929} C_VEL
LIN {X 0,Y 63.413,Z 526.81,A -85,B 0,C 180,E1 26009.968,E2 26009.968} C_VEL
LIN {X 0,Y 60.785,Z 526.81,A -85,B 0,C 180,E1 26024.389,E2 26024.389} C_VEL
LIN {X 0,Y 58.123,Z 526.81,A -85,B 0,C 180,E1 26048.534,E2 26048.534} C_VEL
LIN {X 0,Y 58.578,Z 526.81,A -85,B 0,C 180,E1 26068.821,E2 26068.821} C_VEL
LIN {X 0,Y 61.502,Z 526.81,A -85,B 0,C 180,E1 26089.782,E2 26089.782} C_VEL
LIN {X 0,Y 63.379,Z 526.81,A -85,B 0,C 180,E1 26099.958,E2 26099.958} C_VEL
LIN {X 0,Y 60.944,Z 526.81,A -85,B 0,C 180,E1 26114.339,E2 26114.339} C_VEL
LIN {X 0,Y 60.171,Z 526.81,A -85,B 0,C 180,E1 26129.643,E2 26129.643} C_VEL
LIN {X 0,Y 71.971,Z 579.243,A -85,B 0,C 180,E1 26143.598,E2 26143.598} C_VEL
LIN {X 0,Y 81.259,Z 612.741,A -85,B 0,C 180,E1 26154.198,E2 26154.198} C_VEL
LIN {X 0,Y 80.821,Z 614.662,A -85,B 0,C 180,E1 26154.968,E2 26154.968} C_VEL
LIN {X 0,Y 76.385,Z 624.854,A -85,B 0,C 180,E1 26160.058,E2 26160.058} C_VEL
LIN {X 0,Y 69.165,Z 640.181,A -85,B 0,C 180,E1 26171.254,E2 26171.254} C_VEL
LIN {X 0,Y 71.026,Z 662.67,A -85,B 0,C 180,E1 26191.17,E2 26191.17} C_VEL
LIN {X 0,Y 72.523,Z 667.519,A -85,B 0,C 180,E1 26196.749,E2 26196.749} C_VEL
LIN {X 0,Y 74.398,Z 675.356,A -85,B 0,C 180,E1 26227.662,E2 26227.662} C_VEL
LIN {X 0,Y 82.139,Z 677.099,A -85,B 0,C 180,E1 26240.504,E2 26240.504} C_VEL
LIN {X 0,Y 67.183,Z 655.701,A -85,B 0,C 180,E1 26260.285,E2 26260.285} C_VEL
LIN {X 0,Y 62.593,Z 630.817,A -85,B 0,C 180,E1 26281.775,E2 26281.775} C_VEL
LIN {X 0,Y 64.589,Z 601.872,A -85,B 0,C 180,E1 26300,E2 26300} C_VEL
LIN {X 0,Y 65.516,Z 589.514,A -85,B 0,C 180,E1 26305.586,E2 26305.586} C_VEL
LIN {X 0,Y 58.837,Z 557.431,A -85,B 0,C 180,E1 26317.258,E2 26317.258} C_VEL
LIN {X 0,Y 51.225,Z 526.81,A -85,B 0,C 180,E1 26328.474,E2 26328.474} C_VEL
LIN {X 0,Y 52.101,Z 526.81,A -85,B 0,C 180,E1 26353.065,E2 26353.065} C_VEL
LIN {X 0,Y 55.267,Z 526.81,A -85,B 0,C 180,E1 26369.963,E2 26369.963} C_VEL
LIN {X 0,Y 52.007,Z 526.81,A -85,B 0,C 180,E1 26386.884,E2 26386.884} C_VEL
LIN {X 0,Y 50.235,Z 526.81,A -85,B 0,C 180,E1 26407.019,E2 26407.019} C_VEL
LIN {X 0,Y 50.232,Z 526.81,A -85,B 0,C 180,E1 26422.863,E2 26422.863} C_VEL
LIN {X 0,Y 51.973,Z 526.81,A -85,B 0,C 180,E1 26443.01,E2 26443.01} C_VEL
LIN {X 0,Y 55.23,Z 526.81,A -85,B 0,C 180,E1 26459.952,E2 26459.952} C_VEL
LIN {X 0,Y 52.279,Z 527.289,A -85,B 0,C 180,E1 26487.493,E2 26487.493} C_VEL
LIN {X 0,Y 63.639,Z 578.328,A -85,B 0,C 180,E1 26503.097,E2 26503.097} C_VEL
LIN {X 0,Y 72.981,Z 611.189,A -85,B 0,C 180,E1 26514.578,E2 26514.578} C_VEL
LIN {X 0,Y 69.456,Z 636.208,A -85,B 0,C 180,E1 26528.448,E2 26528.448} C_VEL
LIN {X 0,Y 69.165,Z 640.181,A -85,B 0,C 180,E1 26531.254,E2 26531.254} C_VEL
LIN {X 0,Y 66.799,Z 648.732,A -85,B 0,C 180,E1 26539.428,E2 26539.428} C_VEL
LIN {X 0,Y 65.136,Z 660.806,A -85,B 0,C 180,E1 26555.579,E2 26555.579} C_VEL
LIN {X 0,Y 65.664,Z 663.618,A -85,B 0,C 180,E1 26559.99,E2 26559.99} C_VEL
LIN {X 0,Y 71.431,Z 671.611,A -85,B 0,C 180,E1 26595.131,E2 26595.131} C_VEL
LIN {X 0,Y 73.374,Z 671.684,A -85,B 0,C 180,E1 26599.456,E2 26599.456} C_VEL
LIN {X 0,Y 58.85,Z 648.737,A -85,B 0,C 180,E1 26621.29,E2 26621.29} C_VEL
LIN {X 0,Y 55.154,Z 623.605,A -85,B 0,C 180,E1 26643.984,E2 26643.984} C_VEL
LIN {X 0,Y 57.908,Z 593.088,A -85,B 0,C 180,E1 26663.5,E2 26663.5} C_VEL
LIN {X 0,Y 52.182,Z 564.214,A -85,B 0,C 180,E1 26675.784,E2 26675.784} C_VEL
LIN {X 0,Y 43.836,Z 529.834,A -85,B 0,C 180,E1 26689.353,E2 26689.353} C_VEL
LIN {X 0,Y 43.116,Z 526.81,A -85,B 0,C 180,E1 26691.581,E2 26691.581} C_VEL
LIN {X 0,Y 43.589,Z 526.81,A -85,B 0,C 180,E1 26709.624,E2 26709.624} C_VEL
LIN {X 0,Y 46.863,Z 526.81,A -85,B 0,C 180,E1 26729.956,E2 26729.956} C_VEL
LIN {X 0,Y 43.368,Z 526.81,A -85,B 0,C 180,E1 26750.383,E2 26750.383} C_VEL
LIN {X 0,Y 41.886,Z 526.81,A -85,B 0,C 180,E1 26776.227,E2 26776.227} C_VEL
LIN {X 0,Y 43.343,Z 526.81,A -85,B 0,C 180,E1 26799.489,E2 26799.489} C_VEL
LIN {X 0,Y 46.821,Z 526.81,A -85,B 0,C 180,E1 26819.943,E2 26819.943} C_VEL
LIN {X 0,Y 44.337,Z 526.94,A -85,B 0,C 180,E1 26844.409,E2 26844.409} C_VEL
LIN {X 0,Y 55.228,Z 577.198,A -85,B 0,C 180,E1 26862.526,E2 26862.526} C_VEL
LIN {X 0,Y 65.049,Z 611.114,A -85,B 0,C 180,E1 26875.828,E2 26875.828} C_VEL
LIN {X 0,Y 62.024,Z 636.64,A -85,B 0,C 180,E1 26892.268,E2 26892.268} C_VEL
LIN {X 0,Y 64.47,Z 658.838,A -85,B 0,C 180,E1 26913.398,E2 26913.398} C_VEL
LIN {X 0,Y 65.136,Z 660.806,A -85,B 0,C 180,E1 26915.579,E2 26915.579} C_VEL
LIN {X 0,Y 64.131,Z 662.911,A -85,B 0,C 180,E1 26921.261,E2 26921.261} C_VEL
LIN {X 0,Y 59.033,Z 662.609,A -85,B 0,C 180,E1 26936.777,E2 26936.777} C_VEL
LIN {X 0,Y 64.823,Z 666.339,A -85,B 0,C 180,E1 26955.577,E2 26955.577} C_VEL
LIN {X 0,Y 65.043,Z 665.863,A -85,B 0,C 180,E1 26957.94,E2 26957.94} C_VEL
LIN {X 0,Y 50.703,Z 641.002,A -85,B 0,C 180,E1 26982.682,E2 26982.682} C_VEL
LIN {X 0,Y 47.887,Z 614.075,A -85,B 0,C 180,E1 27008.007,E2 27008.007} C_VEL
LIN {X 0,Y 49.76,Z 590.402,A -85,B 0,C 180,E1 27024,E2 27024} C_VEL
LIN {X 0,Y 42.722,Z 557.5,A -85,B 0,C 180,E1 27039.733,E2 27039.733} C_VEL
LIN {X 0,Y 35.043,Z 526.81,A -85,B 0,C 180,E1 27055.83,E2 27055.83} C_VEL
LIN {X 0,Y 38.487,Z 526.81,A -85,B 0,C 180,E1 27089.947,E2 27089.947} C_VEL
LIN {X 0,Y 34.157,Z 526.81,A -85,B 0,C 180,E1 27117.395,E2 27117.395} C_VEL
LIN {X 0,Y 33.78,Z 526.81,A -85,B 0,C 180,E1 27130.837,E2 27130.837} C_VEL
LIN {X 0,Y 34.268,Z 526.81,A -85,B 0,C 180,E1 27153.694,E2 27153.694} C_VEL
LIN {X 0,Y 38.44,Z 526.81,A -85,B 0,C 180,E1 27179.93,E2 27179.93} C_VEL
LIN {X 0,Y 36.524,Z 527.398,A -85,B 0,C 180,E1 27200.599,E2 27200.599} C_VEL
LIN {X 0,Y 46.781,Z 575.698,A -85,B 0,C 180,E1 27221.798,E2 27221.798} C_VEL
LIN {X 0,Y 56.939,Z 610.214,A -85,B 0,C 180,E1 27237.182,E2 27237.182} C_VEL
LIN {X 0,Y 55.008,Z 631.124,A -85,B 0,C 180,E1 27252.001,E2 27252.001} C_VEL
LIN {X 0,Y 57.41,Z 652.841,A -85,B 0,C 180,E1 27273.816,E2 27273.816} C_VEL
LIN {X 0,Y 59.45,Z 658.641,A -85,B 0,C 180,E1 27281.047,E2 27281.047} C_VEL
LIN {X 0,Y 59.033,Z 662.609,A -85,B 0,C 180,E1 27296.777,E2 27296.777} C_VEL
LIN {X 0,Y 57.286,Z 661.36,A -85,B 0,C 180,E1 27303.321,E2 27303.321} C_VEL
LIN {X 0,Y 55.96,Z 659.56,A -85,B 0,C 180,E1 27310.362,E2 27310.362} C_VEL
LIN {X 0,Y 57.374,Z 659.955,A -85,B 0,C 180,E1 27315.466,E2 27315.466} C_VEL
LIN {X 0,Y 43.227,Z 634.37,A -85,B 0,C 180,E1 27342.219,E2 27342.219} C_VEL
LIN {X 0,Y 40.721,Z 606.26,A -85,B 0,C 180,E1 27370.78,E2 27370.78} C_VEL
LIN {X 0,Y 41.68,Z 589.998,A -85,B 0,C 180,E1 27383.017,E2 27383.017} C_VEL
LIN {X 0,Y 34.72,Z 557.761,A -85,B 0,C 180,E1 27401.363,E2 27401.363} C_VEL
LIN {X 0,Y 27.821,Z 530.073,A -85,B 0,C 180,E1 27419.237,E2 27419.237} C_VEL
LIN {X 0,Y 27.18,Z 526.81,A -85,B 0,C 180,E1 27423.004,E2 27423.004} C_VEL
LIN {X 0,Y 29.644,Z 526.81,A -85,B 0,C 180,E1 27449.931,E2 27449.931} C_VEL
LIN {X 0,Y 25.818,Z 526.81,A -85,B 0,C 180,E1 27485.806,E2 27485.806} C_VEL
LIN {X 0,Y 25.505,Z 526.81,A -85,B 0,C 180,E1 27503.456,E2 27503.456} C_VEL
LIN {X 0,Y 29.584,Z 526.81,A -85,B 0,C 180,E1 27539.91,E2 27539.91} C_VEL
LIN {X 0,Y 28.796,Z 527.576,A -85,B 0,C 180,E1 27554.789,E2 27554.789} C_VEL
LIN {X 0,Y 38.574,Z 574.999,A -85,B 0,C 180,E1 27581.385,E2 27581.385} C_VEL
LIN {X 0,Y 49.245,Z 610.418,A -85,B 0,C 180,E1 27599.739,E2 27599.739} C_VEL
LIN {X 0,Y 48.236,Z 634.674,A -85,B 0,C 180,E1 27621.014,E2 27621.014} C_VEL
LIN {X 0,Y 53.018,Z 653.053,A -85,B 0,C 180,E1 27642.407,E2 27642.407} C_VEL
LIN {X 0,Y 54.31,Z 658.44,A -85,B 0,C 180,E1 27663.933,E2 27663.933} C_VEL
LIN {X 0,Y 55.96,Z 659.56,A -85,B 0,C 180,E1 27670.362,E2 27670.362} C_VEL
LIN {X 0,Y 54.346,Z 657.207,A -85,B 0,C 180,E1 27674.947,E2 27674.947} C_VEL
LIN {X 0,Y 42.597,Z 643.017,A -85,B 0,C 180,E1 27682.661,E2 27682.661} C_VEL
LIN {X 0,Y 33.765,Z 617.012,A -85,B 0,C 180,E1 27713.644,E2 27713.644} C_VEL
LIN {X 0,Y 33.86,Z 590.182,A -85,B 0,C 180,E1 27740.904,E2 27740.904} C_VEL
LIN {X 0,Y 26.711,Z 558.03,A -85,B 0,C 180,E1 27763.689,E2 27763.689} C_VEL
LIN {X 0,Y 20.964,Z 532.892,A -85,B 0,C 180,E1 27785.923,E2 27785.923} C_VEL
LIN {X 0,Y 19.653,Z 526.81,A -85,B 0,C 180,E1 27795.961,E2 27795.961} C_VEL
LIN {X 0,Y 20.533,Z 526.81,A -85,B 0,C 180,E1 27809.9,E2 27809.9} C_VEL
LIN {X 0,Y 17.794,Z 526.81,A -85,B 0,C 180,E1 27841.41,E2 27841.41} C_VEL
LIN {X 0,Y 17.501,Z 526.81,A -85,B 0,C 180,E1 27869.666,E2 27869.666} C_VEL
LIN {X 0,Y 21.201,Z 526.81,A -85,B 0,C 180,E1 27903.712,E2 27903.712} C_VEL
LIN {X 0,Y 27.167,Z 559.72,A -85,B 0,C 180,E1 27931.383,E2 27931.383} C_VEL
LIN {X 0,Y 36.773,Z 596.897,A -85,B 0,C 180,E1 27955.3,E2 27955.3} C_VEL
LIN {X 0,Y 41.816,Z 611.635,A -85,B 0,C 180,E1 27964.184,E2 27964.184} C_VEL
LIN {X 0,Y 42.818,Z 637.365,A -85,B 0,C 180,E1 27992.353,E2 27992.353} C_VEL
LIN {X 0,Y 47.515,Z 649.389,A -85,B 0,C 180,E1 28008.627,E2 28008.627} C_VEL
LIN {X 0,Y 49.398,Z 653.079,A -85,B 0,C 180,E1 28029.75,E2 28029.75} C_VEL
LIN {X 0,Y 49.521,Z 652.781,A -85,B 0,C 180,E1 28032.837,E2 28032.837} C_VEL
LIN {X 0,Y 42.597,Z 643.017,A -85,B 0,C 180,E1 28042.661,E2 28042.661} C_VEL
LIN {X 0,Y 36.352,Z 632.99,A -85,B 0,C 180,E1 28050.646,E2 28050.646} C_VEL
LIN {X 0,Y 27.752,Z 616.421,A -85,B 0,C 180,E1 28063.873,E2 28063.873} C_VEL
LIN {X 0,Y 27.309,Z 614.556,A -85,B 0,C 180,E1 28066.351,E2 28066.351} C_VEL
LIN {X 0,Y 25.971,Z 589.819,A -85,B 0,C 180,E1 28097.66,E2 28097.66} C_VEL
LIN {X 0,Y 18.85,Z 558.646,A -85,B 0,C 180,E1 28127.185,E2 28127.185} C_VEL
LIN {X 0,Y 14.446,Z 534.595,A -85,B 0,C 180,E1 28160.431,E2 28160.431} C_VEL
LIN {X 0,Y 13.415,Z 531.74,A -85,B 0,C 180,E1 28169.847,E2 28169.847} C_VEL
LIN {X 0,Y 11.056,Z 531.844,A -85,B 0,C 180,E1 28221.83,E2 28221.83} C_VEL
LIN {X 0,Y 15.683,Z 534.057,A -85,B 0,C 180,E1 28257.707,E2 28257.707} C_VEL
LIN {X 0,Y 22.745,Z 576.314,A -85,B 0,C 180,E1 28303.188,E2 28303.188} C_VEL
LIN {X 0,Y 34.298,Z 609.966,A -85,B 0,C 180,E1 28328.279,E2 28328.279} C_VEL
LIN {X 0,Y 37.195,Z 634.097,A -85,B 0,C 180,E1 28358.836,E2 28358.836} C_VEL
LIN {X 0,Y 41.64,Z 643.416,A -85,B 0,C 180,E1 28371.375,E2 28371.375} C_VEL
LIN {X 0,Y 42.446,Z 645.586,A -85,B 0,C 180,E1 28379.536,E2 28379.536} C_VEL
LIN {X 0,Y 42.606,Z 645.721,A -85,B 0,C 180,E1 28388.652,E2 28388.652} C_VEL
LIN {X 0,Y 28.605,Z 619.954,A -85,B 0,C 180,E1 28418.762,E2 28418.762} C_VEL
LIN {X 0,Y 27.309,Z 614.556,A -85,B 0,C 180,E1 28426.351,E2 28426.351} C_VEL
LIN {X 0,Y 24.009,Z 603.142,A -85,B 0,C 180,E1 28439.062,E2 28439.062} C_VEL
LIN {X 0,Y 16.422,Z 583.012,A -85,B 0,C 180,E1 28458.735,E2 28458.735} C_VEL
LIN {X 0,Y 10.222,Z 551.249,A -85,B 0,C 180,E1 28510.882,E2 28510.882} C_VEL
LIN {X 0,Y 9.532,Z 538.906,A -85,B 0,C 180,E1 28546.594,E2 28546.594} C_VEL
LIN {X 0,Y 10.269,Z 540.296,A -85,B 0,C 180,E1 28600.872,E2 28600.872} C_VEL
LIN {X 0,Y 15.215,Z 578.196,A -85,B 0,C 180,E1 28668.008,E2 28668.008} C_VEL
LIN {X 0,Y 27.559,Z 610.24,A -85,B 0,C 180,E1 28696.992,E2 28696.992} C_VEL
LIN {X 0,Y 33.993,Z 634.064,A -85,B 0,C 180,E1 28732.263,E2 28732.263} C_VEL
LIN {X 0,Y 37.266,Z 639.309,A -85,B 0,C 180,E1 28739.807,E2 28739.807} C_VEL
LIN {X 0,Y 32.974,Z 633.778,A -85,B 0,C 180,E1 28746.669,E2 28746.669} C_VEL
LIN {X 0,Y 20.181,Z 606.472,A -85,B 0,C 180,E1 28783.799,E2 28783.799} C_VEL
LIN {X 0,Y 18.491,Z 590.002,A -85,B 0,C 180,E1 28810.621,E2 28810.621} C_VEL
LIN {X 0,Y 16.422,Z 583.012,A -85,B 0,C 180,E1 28818.735,E2 28818.735} C_VEL
LIN {X 0,Y 11.106,Z 571.568,A -85,B 0,C 180,E1 28834.048,E2 28834.048} C_VEL
LIN {X 0,Y 5.391,Z 552.854,A -85,B 0,C 180,E1 28918.94,E2 28918.94} C_VEL
LIN {X 0,Y 5.81,Z 551.24,A -85,B 0,C 180,E1 28933.621,E2 28933.621} C_VEL
LIN {X 0,Y 10.82,Z 587.227,A -85,B 0,C 180,E1 29053.273,E2 29053.273} C_VEL
LIN {X 0,Y 21.573,Z 609.572,A -85,B 0,C 180,E1 29070.095,E2 29070.095} C_VEL
LIN {X 0,Y 27.186,Z 624.958,A -85,B 0,C 180,E1 29095.429,E2 29095.429} C_VEL
LIN {X 0,Y 25.255,Z 622.506,A -85,B 0,C 180,E1 29100.693,E2 29100.693} C_VEL
LIN {X 0,Y 12.426,Z 593.679,A -85,B 0,C 180,E1 29147.015,E2 29147.015} C_VEL
LIN {X 0,Y 9.483,Z 584.266,A -85,B 0,C 180,E1 29162.48,E2 29162.48} C_VEL
LIN {X 0,Y 5.391,Z 552.854,A -85,B 0,C 180,E1 29278.94,E2 29278.94} C_VEL
LIN {X 0,Y 8.104,Z 553.632,A -85,B 0,C 180,E1 29302.696,E2 29302.696} C_VEL
LIN {X 0,Y 8.104,Z 779,A -85,B 0,C 180,E1 29302.696,E2 29302.696} C_VEL
LIN {X 0,Y 8.104,Z 779,A -85,B 0,C 180,E1 29302.696,E2 29302.696}

